  MoveL 2052 to (224.55, 431.71, -17.53) mm, rotated rx -180 ry 0 rz -11.91 deg; joints [23.109, -21.337, 64.711, -81.9, 97.908, 133.105]
  MoveL 2053 to (224.32, 431.8, -17.52) mm, rotated rx -180 ry 0 rz -11.91 deg; joints [23.101, -21.338, 64.711, -81.906, 97.902, 133.105]
  MoveL 2054 to (224.09, 431.88, -17.52) mm, rotated rx -180 ry 0 rz -11.91 deg; joints [23.094, -21.339, 64.715, -81.911, 97.897, 133.106]
  MoveL 2055 to (224.01, 431.9, -17.53) mm, rotated rx -180 ry 0 rz -11.91 deg; joints [23.091, -21.34, 64.716, -81.912, 97.895, 133.106]
  MoveL 2056 to (223.77, 431.95, -17.53) mm, rotated rx -180 ry 0 rz -11.91 deg; joints [23.084, -21.343, 64.723, -81.917, 97.889, 133.109]
  MoveL 2057 to (223.53, 431.98, -17.53) mm, rotated rx -180 ry 0 rz -11.91 deg; joints [23.076, -21.347, 64.733, -81.921, 97.883, 133.114]
  MoveL 2058 to (223.29, 431.99, -17.53) mm, rotated rx -180 ry 0 rz -11.91 deg; joints [23.069, -21.353, 64.745, -81.925, 97.877, 133.119]
  MoveL 2059 to (223.05, 431.99, -17.53) mm, rotated rx 180 ry 0 rz -11.91 deg; joints [23.062, -21.359, 64.759, -81.929, 97.871, 133.126]
  MoveL 2060 to (-164.9, 431.99, -17.53) mm, rotated rx 180 ry 0 rz -11.91 deg; joints [11.107, -28.262, 79.844, -90.307, 89.248, 140.713]
  MoveL 2061 to (-194.97, 431.99, -17.52) mm, rotated rx -180 ry 0 rz -11.91 deg; joints [10.122, -28.555, 80.501, -91.087, 88.643, 141.084]
  MoveL 2062 to (-195.47, 431.99, -17.53) mm, rotated rx -180 ry 0 rz -11.91 deg; joints [10.106, -28.56, 80.512, -91.1, 88.633, 141.09]
  Set speed (38.1 mm/s)
  MoveL 2063 to (-196.09, 432.77, -17.53) mm, rotated rx -180 ry 0 rz -11.91 deg; joints [10.081, -28.525, 80.435, -91.119, 88.617, 141.049]
  MoveL 2064 to (-195.65, 434.72, -17.53) mm, rotated rx 180 ry 0 rz -11.91 deg; joints [10.084, -28.417, 80.2, -91.113, 88.616, 140.922]
  MoveL 2065 to (-195.51, 435.34, -16.89) mm, rotated rx 180 ry 0 rz -11.91 deg; joints [10.084, -28.412, 80.132, -91.111, 88.615, 140.859]
  Set speed (100.0 mm/s)
  MoveL 2066 to (-195.51, 435.34, 34.53) mm, rotated rx -180 ry 0 rz -11.91 deg; joints [10.073, -30.771, 80.586, -91.073, 88.572, 138.953]
  MoveL 2067 to (-195.51, 435.34, 34.53) mm, rotated rx -180 ry 0 rz -11.91 deg; joints [10.073, -30.771, 80.586, -91.073, 88.572, 138.953]

--- program Machining (robot KUKA KR 30 HA) ---
  Smooth(1)
  Print: /'1001'
  Print: /''
  Print: /'Parallel1'
  Call SetTool(1)
  Call SetRPM(5000.0)
  Set speed (1000.0 mm/s)
  Set Ref.: Frame 4
  Set Tool: rc90 spindle mm
  Show rc90 spindle mm
  MoveJ 1 to (194.72, 277.93, 99.72) mm, rotated rx -149.92 ry 0.28 rz 179.52 deg; joints [9.071, -45.044, 108.371, -170.24, 63.004, 205.935]
  MoveL 2 to (194.72, 277.93, 99.72) mm, rotated rx -149.92 ry 0.28 rz 179.52 deg; joints [9.071, -45.044, 108.371, -170.24, 63.004, 205.935]
  MoveL 3 to (194.72, 227.8, 13.19) mm, rotated rx -149.92 ry 0.28 rz 179.52 deg; joints [11.04, -39.933, 106.924, -168.39, 66.758, 205.788]
  MoveL 4 to (194.72, 227.8, 13.19) mm, rotated rx -149.92 ry 0.28 rz 179.52 deg; joints [11.04, -39.933, 106.924, -168.39, 66.758, 205.788]
  Set speed (1000.0 mm/s)
  MoveL 5 to (194.72, 218.79, -2.36) mm, rotated rx -149.92 ry 0.28 rz 179.52 deg; joints [11.391, -38.991, 106.584, -168.061, 67.374, 205.777]
  Set speed (16.7 mm/s)
  MoveL 6 to (194.72, 209.92, -17.68) mm, rotated rx -149.92 ry 0.28 rz 179.52 deg; joints [11.737, -38.057, 106.224, -167.738, 67.963, 205.769]
  MoveL 7 to (193.72, 209.42, -18.55) mm, rotated rx -149.92 ry 0.28 rz 179.52 deg; joints [11.765, -38.04, 106.292, -167.716, 68.048, 205.778]
  MoveL 8 to (193.59, 214.43, -9.89) mm, rotated rx -149.92 ry 0.28 rz 179.52 deg; joints [11.57, -38.574, 106.51, -167.897, 67.725, 205.783]
  MoveL 9 to (193.59, 214.44, -9.88) mm, rotated rx -149.92 ry 0.28 rz 179.52 deg; joints [11.57, -38.574, 106.51, -167.898, 67.724, 205.783]
  Set speed (1000.0 mm/s)
  MoveL 10 to (193.59, 222.79, 4.53) mm, rotated rx -149.92 ry 0.28 rz 179.52 deg; joints [11.244, -39.451, 106.838, -168.202, 67.161, 205.791]
  MoveL 11 to (194.72, 224.52, 3.53) mm, rotated rx -149.92 ry 0.28 rz 179.52 deg; joints [11.169, -39.365, 106.757, -168.284, 67.16, 205.822]
  MoveL 12 to (194.72, 217.03, -9.4) mm, rotated rx -149.92 ry 0.28 rz 179.52 deg; joints [11.461, -38.579, 106.464, -168.011, 67.665, 205.814]
  Set speed (16.7 mm/s)
  MoveL 13 to (194.72, 211.65, -18.68) mm, rotated rx -149.92 ry 0.28 rz 179.52 deg; joints [11.671, -38.012, 106.243, -167.815, 68.02, 205.81]
  MoveC 14 to (194.43, 211.3, -19.3) mm, rotated rx -149.92 ry 0.28 rz 179.52 deg; joints [11.687, -37.985, 106.254, -167.8, 68.058, 205.812] to (193.72, 211.15, -19.55) mm, rotated rx -149.92 ry 0.28 rz 179.52 deg; joints [11.698, -37.995, 106.31, -167.792, 68.105, 205.818]
  MoveL 15 to (193.72, 211.15, -19.55) mm, rotated rx -149.92 ry 0.28 rz 179.52 deg; joints [11.698, -37.995, 106.31, -167.792, 68.105, 205.818]
  MoveL 16 to (193.49, 216.16, -10.9) mm, rotated rx -149.92 ry 0.28 rz 179.52 deg; joints [11.505, -38.533, 106.538, -167.974, 67.787, 205.824]
  MoveL 17 to (191.2, 216.16, -10.9) mm, rotated rx -149.92 ry 0.28 rz 179.52 deg; joints [11.523, -38.615, 106.74, -167.965, 67.905, 205.844]
  MoveC 18 to (190.5, 216.31, -10.64) mm, rotated rx -149.92 ry 0.28 rz 179.52 deg; joints [11.523, -38.656, 106.808, -167.967, 67.932, 205.85] to (190.2, 216.66, -10.03) mm, rotated rx -149.92 ry 0.28 rz 179.52 deg; joints [11.511, -38.704, 106.848, -167.979, 67.923, 205.853]
  MoveL 19 to (190.2, 216.66, -10.03) mm, rotated rx -149.92 ry 0.28 rz 179.52 deg; joints [11.511, -38.704, 106.848, -167.979, 67.923, 205.853]
  Set speed (1000.0 mm/s)
  MoveL 20 to (190.2, 224.52, 3.53) mm, rotated rx -149.92 ry 0.28 rz 179.52 deg; joints [11.204, -39.531, 107.156, -168.266, 67.392, 205.86]
  MoveL 21 to (-191.54, 222.79, 4.53) mm, rotated rx -149.92 ry 0.28 rz 179.52 deg; joints [15.261, -50.505, 137.346, -165.09, 86.292, 209.487]
  MoveL 22 to (-191.54, 219.49, -1.15) mm, rotated rx -149.92 ry 0.28 rz 179.52 deg; joints [15.432, -50.022, 137.196, -164.925, 86.617, 209.565]
  Set speed (16.7 mm/s)
  MoveL 23 to (-191.54, 214.63, -9.56) mm, rotated rx -149.92 ry 0.28 rz 179.52 deg; joints [15.684, -49.309, 136.968, -164.679, 87.087, 209.681]
  MoveL 24 to (-191.94, 214.43, -9.89) mm, rotated rx -149.92 ry 0.28 rz 179.52 deg; joints [15.699, -49.288, 136.987, -164.664, 87.126, 209.691]
  MoveL 25 to (-192.68, 214.43, -9.89) mm, rotated rx -149.92 ry 0.28 rz 179.52 deg; joints [15.71, -49.302, 137.04, -164.654, 87.164, 209.702]
  MoveL 26 to (-192.7, 209.42, -18.55) mm, rotated rx -149.92 ry 0.28 rz 179.52 deg; joints [15.969, -48.568, 136.797, -164.401, 87.639, 209.824]
  MoveL 27 to (-193.07, 211.15, -19.55) mm, rotated rx -149.92 ry 0.28 rz 179.52 deg; joints [15.887, -48.5, 136.842, -164.484, 87.747, 209.856]
  MoveL 28 to (-193.07, 216.16, -10.9) mm, rotated rx -149.92 ry 0.28 rz 179.52 deg; joints [15.628, -49.234, 137.086, -164.738, 87.273, 209.735]
  MoveL 29 to (-189.43, 216.16, -10.9) mm, rotated rx -149.92 ry 0.28 rz 179.52 deg; joints [15.576, -49.167, 136.825, -164.787, 87.086, 209.686]
  MoveL 30 to (-188.93, 216.41, -10.46) mm, rotated rx -149.92 ry 0.28 rz 179.52 deg; joints [15.556, -49.194, 136.801, -164.807, 87.037, 209.673]
  MoveC 31 to (-189.34, 217.09, -9.63) mm, rotated rx -149.92 ry 0.28 rz 179.52 deg; joints [15.527, -49.273, 136.858, -164.835, 87.014, 209.668] to (-190.32, 217.64, -9.44) mm, rotated rx -149.92 ry 0.28 rz 179.52 deg; joints [15.513, -49.309, 136.942, -164.851, 87.061, 209.682]
  MoveL 32 to (-190.32, 217.64, -9.44) mm, rotated rx -149.92 ry 0.28 rz 179.52 deg; joints [15.513, -49.309, 136.942, -164.851, 87.061, 209.682]
  MoveL 33 to (-192.56, 218.42, -9.89) mm, rotated rx -149.92 ry 0.28 rz 179.52 deg; joints [15.505, -49.318, 137.111, -164.86, 87.215, 209.724]
  MoveC 34 to (-193.55, 218.53, -10.47) mm, rotated rx -149.92 ry 0.28 rz 179.52 deg; joints [15.513, -49.289, 137.175, -164.853, 87.305, 209.748] to (-193.96, 218.14, -11.47) mm, rotated rx -149.92 ry 0.28 rz 179.52 deg; joints [15.54, -49.213, 137.18, -164.828, 87.384, 209.768]
  MoveL 35 to (-193.96, 218.14, -11.47) mm, rotated rx -149.92 ry 0.28 rz 179.52 deg; joints [15.54, -49.213, 137.18, -164.828, 87.384, 209.768]
  MoveL 36 to (-193.96, 213.13, -20.12) mm, rotated rx -149.92 ry 0.28 rz 179.52 deg; joints [15.799, -48.478, 136.935, -164.573, 87.859, 209.89]
  MoveL 37 to (-193.46, 212.88, -20.55) mm, rotated rx -149.92 ry 0.28 rz 179.52 deg; joints [15.805, -48.432, 136.887, -164.567, 87.856, 209.889]
  MoveL 38 to (-193.43, 217.89, -11.9) mm, rotated rx -149.92 ry 0.28 rz 179.52 deg; joints [15.545, -49.166, 137.131, -164.822, 87.381, 209.767]
  MoveL 39 to (193.49, 217.89, -11.9) mm, rotated rx -149.92 ry 0.28 rz 179.52 deg; joints [11.438, -38.488, 106.556, -168.051, 67.843, 205.865]
  MoveL 40 to (193.72, 212.88, -20.55) mm, rotated rx -149.92 ry 0.28 rz 179.52 deg; joints [11.632, -37.95, 106.328, -167.869, 68.161, 205.858]
  MoveL 41 to (193.72, 214.61, -21.55) mm, rotated rx -149.92 ry 0.28 rz 179.52 deg; joints [11.566, -37.905, 106.346, -167.945, 68.218, 205.898]
  MoveL 42 to (193.49, 219.62, -12.9) mm, rotated rx -149.92 ry 0.28 rz 179.52 deg; joints [11.372, -38.442, 106.574, -168.128, 67.9, 205.905]
  MoveL 43 to (-193.72, 219.62, -12.9) mm, rotated rx -149.92 ry 0.28 rz 179.52 deg; joints [15.461, -49.097, 137.169, -164.907, 87.485, 209.798]
  MoveL 44 to (-193.74, 214.61, -21.55) mm, rotated rx -149.92 ry 0.28 rz 179.52 deg; joints [15.721, -48.362, 136.925, -164.652, 87.96, 209.92]
  MoveL 45 to (-193.31, 216.34, -22.56) mm, rotated rx -149.92 ry 0.28 rz 179.52 deg; joints [15.627, -48.28, 136.912, -164.747, 88.026, 209.94]
  MoveL 46 to (-193.31, 221.35, -13.9) mm, rotated rx -149.92 ry 0.28 rz 179.52 deg; joints [15.367, -49.014, 137.158, -165.002, 87.552, 209.82]
  MoveL 47 to (193.28, 221.35, -13.9) mm, rotated rx -149.92 ry 0.28 rz 179.52 deg; joints [11.307, -38.405, 106.61, -168.204, 67.967, 205.947]
  MoveL 48 to (193.31, 216.34, -22.56) mm, rotated rx -149.92 ry 0.28 rz 179.52 deg; joints [11.502, -37.874, 106.399, -168.02, 68.295, 205.942]
  MoveL 49 to (191.75, 218.07, -23.56) mm, rotated rx -149.92 ry 0.28 rz 179.52 deg; joints [11.448, -37.884, 106.555, -168.09, 68.433, 205.995]
  MoveL 50 to (191.68, 223.08, -14.91) mm, rotated rx -149.92 ry 0.28 rz 179.52 deg; joints [11.253, -38.416, 106.768, -168.274, 68.107, 206]
  MoveL 51 to (-191.75, 223.08, -14.91) mm, rotated rx -149.92 ry 0.28 rz 179.52 deg; joints [15.257, -48.911, 137.063, -165.112, 87.56, 209.825]
  MoveL 52 to (-191.75, 218.07, -23.56) mm, rotated rx -149.92 ry 0.28 rz 179.52 deg; joints [15.517, -48.177, 136.817, -164.857, 88.033, 209.945]
  MoveC 53 to (-192.46, 218.22, -23.31) mm, rotated rx -149.92 ry 0.28 rz 179.52 deg; joints [15.519, -48.211, 136.875, -164.855, 88.056, 209.951] to (-192.75, 218.57, -22.69) mm, rotated rx -149.92 ry 0.28 rz 179.52 deg; joints [15.505, -48.268, 136.914, -164.869, 88.038, 209.947]
  MoveL 54 to (-192.75, 218.57, -22.69) mm, rotated rx -149.92 ry 0.28 rz 179.52 deg; joints [15.505, -48.268, 136.914, -164.869, 88.038, 209.947]
  Set speed (1000.0 mm/s)
  MoveL 55 to (-192.75, 236.46, 8.18) mm, rotated rx -149.92 ry 0.28 rz 179.52 deg; joints [14.575, -50.894, 137.748, -165.778, 86.296, 209.527]
  Print: /'Parallel2'
  Call SetTool(1)
  Call SetRPM(5000.0)
  Set speed (1000.0 mm/s)
  MoveL 56 to (-122.87, -170.47, 35.88) mm, rotated rx -149.92 ry 0.28 rz 179.52 deg; joints [31.344, -46.991, 120.44, -147.856, 75.214, 201.582]
  MoveL 57 to (-122.87, -192.28, -1.78) mm, rotated rx -149.92 ry 0.28 rz 179.52 deg; joints [32.175, -44.225, 119.07, -147.197, 76.514, 202.158]
  Set speed (16.7 mm/s)
  MoveL 58 to (-122.87, -206.58, -26.46) mm, rotated rx -149.92 ry 0.28 rz 179.52 deg; joints [32.712, -42.414, 118.095, -146.757, 77.289, 202.508]
  MoveC 59 to (-122.57, -206.94, -27.07) mm, rotated rx -149.92 ry 0.28 rz 179.52 deg; joints [32.718, -42.362, 118.05, -146.752, 77.296, 202.51] to (-121.87, -207.08, -27.32) mm, rotated rx -149.92 ry 0.28 rz 179.52 deg; joints [32.707, -42.325, 117.99, -146.76, 77.275, 202.5]
  MoveL 60 to (-121.87, -207.08, -27.32) mm, rotated rx -149.92 ry 0.28 rz 179.52 deg; joints [32.707, -42.325, 117.99, -146.76, 77.275, 202.5]
  MoveL 61 to (-121.78, -193.28, -3.5) mm, rotated rx -149.92 ry 0.28 rz 179.52 deg; joints [32.187, -44.069, 118.928, -147.186, 76.527, 202.162]
  MoveL 62 to (189.07, -193.28, -3.5) mm, rotated rx -149.92 ry 0.28 rz 179.52 deg; joints [26.181, -33.899, 94.323, -150.758, 62.981, 196.347]
  MoveL 63 to (189.08, -207.08, -27.32) mm, rotated rx -149.92 ry 0.28 rz 179.52 deg; joints [26.635, -32.401, 93.386, -150.403, 63.579, 196.439]
  MoveL 64 to (192.38, -208.45, -26.53) mm, rotated rx -149.92 ry 0.28 rz 179.52 deg; joints [26.626, -32.286, 93.034, -150.355, 63.37, 196.312]
  MoveL 65 to (193.72, -211.41, -24.82) mm, rotated rx -149.92 ry 0.28 rz 179.52 deg; joints [26.698, -32.266, 92.801, -150.224, 63.203, 196.16]
  MoveL 66 to (193.72, -197.6, -1) mm, rotated rx -149.92 ry 0.28 rz 179.52 deg; joints [26.246, -33.761, 93.74, -150.576, 62.609, 196.07]
  MoveL 67 to (-126.28, -197.6, -1) mm, rotated rx -149.92 ry 0.28 rz 179.52 deg; joints [32.45, -44.28, 119.084, -146.912, 76.518, 202.072]
  MoveL 68 to (-126.51, -211.41, -24.82) mm, rotated rx -149.92 ry 0.28 rz 179.52 deg; joints [32.973, -42.537, 118.157, -146.485, 77.273, 202.418]
  MoveL 69 to (-126.14, -213.57, -23.57) mm, rotated rx -149.92 ry 0.28 rz 179.52 deg; joints [33.042, -42.574, 118.051, -146.397, 77.164, 202.322]
  MoveL 70 to (-125.68, -215.73, -22.32) mm, rotated rx -149.92 ry 0.28 rz 179.52 deg; joints [33.109, -42.608, 117.94, -146.311, 77.053, 202.226]
  MoveL 71 to (-125.64, -207.44, -8.02) mm, rotated rx -149.92 ry 0.28 rz 179.52 deg; joints [32.799, -43.655, 118.509, -146.563, 76.611, 202.022]
  MoveL 72 to (-121.57, -207.44, -8.02) mm, rotated rx -149.92 ry 0.28 rz 179.52 deg; joints [32.703, -43.547, 118.225, -146.637, 76.45, 201.944]
  MoveL 73 to (-121.42, -201.93, 1.51) mm, rotated rx -149.92 ry 0.28 rz 179.52 deg; joints [32.494, -44.24, 118.584, -146.806, 76.139, 201.803]
  MoveL 74 to (188.78, -201.93, 1.51) mm, rotated rx -149.92 ry 0.28 rz 179.52 deg; joints [26.463, -34.003, 94.024, -150.349, 62.698, 195.987]
  MoveL 75 to (188.9, -207.44, -8.02) mm, rotated rx -149.92 ry 0.28 rz 179.52 deg; joints [26.642, -33.402, 93.646, -150.211, 62.937, 196.024]
  MoveL 76 to (193.72, -207.44, -8.02) mm, rotated rx -149.92 ry 0.28 rz 179.52 deg; joints [26.565, -33.21, 93.208, -150.232, 62.704, 195.925]
  MoveL 77 to (193.72, -215.73, -22.32) mm, rotated rx -149.92 ry 0.28 rz 179.52 deg; joints [26.835, -32.312, 92.638, -150.022, 63.055, 195.977]
  MoveL 78 to (193.72, -217.89, -21.07) mm, rotated rx -149.92 ry 0.28 rz 179.52 deg; joints [26.903, -32.334, 92.555, -149.921, 62.981, 195.885]
  MoveL 79 to (193.7, -220.05, -19.82) mm, rotated rx -149.92 ry 0.28 rz 179.52 deg; joints [26.972, -32.357, 92.474, -149.819, 62.908, 195.793]
  MoveL 80 to (193.7, -211.76, -5.52) mm, rotated rx -149.92 ry 0.28 rz 179.52 deg; joints [26.702, -33.255, 93.044, -150.028, 62.557, 195.74]
  MoveL 81 to (-124.73, -211.76, -5.52) mm, rotated rx -149.92 ry 0.28 rz 179.52 deg; joints [32.934, -43.72, 118.284, -146.388, 76.388, 201.827]
  MoveL 82 to (-124.77, -220.05, -19.82) mm, rotated rx -149.92 ry 0.28 rz 179.52 deg; joints [33.242, -42.674, 117.716, -146.138, 76.83, 202.031]
  MoveC 83 to (-125.47, -219.9, -19.56) mm, rotated rx -149.92 ry 0.28 rz 179.52 deg; joints [33.253, -42.711, 117.776, -146.129, 76.851, 202.041] to (-125.77, -219.55, -18.95) mm, rotated rx -149.92 ry 0.28 rz 179.52 deg; joints [33.247, -42.764, 117.821, -146.134, 76.844, 202.038]
  MoveL 84 to (-125.77, -219.55, -18.95) mm, rotated rx -149.92 ry 0.28 rz 179.52 deg; joints [33.247, -42.764, 117.821, -146.134, 76.844, 202.038]
  Set speed (1000.0 mm/s)
  MoveL 85 to (-125.77, -183.44, 43.39) mm, rotated rx -149.92 ry 0.28 rz 179.52 deg; joints [31.891, -47.334, 120.153, -147.206, 74.768, 201.093]
  Print: /'Contour6'
  Call SetTool(1)
  Call SetRPM(5000.0)
  Set speed (1000.0 mm/s)
  MoveL 86 to (-194.89, 224.1, 15) mm, rotated rx -180 ry 0 rz 179.9 deg; joints [21.967, -53.45, 134.896, -157.76, 81.141, 176.985]
  MoveL 87 to (-194.89, 224.1, 1.16) mm, rotated rx -180 ry 0 rz 179.9 deg; joints [21.974, -52.375, 134.756, -157.806, 82.007, 177.341]
  Set speed (5.6 mm/s)
  MoveL 88 to (-194.89, 224.1, -5) mm, rotated rx -180 ry 0 rz 179.9 deg; joints [21.977, -51.896, 134.688, -157.824, 82.388, 177.498]
  MoveC 89 to (-194.65, 223.92, -5.71) mm, rotated rx 180 ry 0 rz 179.9 deg; joints [21.981, -51.833, 134.658, -157.822, 82.418, 177.51] to (-194.08, 223.5, -6) mm, rotated rx -180 ry 0 rz 179.9 deg; joints [21.99, -51.793, 134.603, -157.812, 82.404, 177.503]
  Set speed (16.7 mm/s)
  MoveL 90 to (-190.41, 220.78, -6) mm, rotated rx 180 ry 0 rz 179.9 deg; joints [22.048, -51.682, 134.266, -157.742, 82.198, 177.41]
  MoveL 91 to (-190.31, 219.26, -6) mm, rotated rx 180 ry 0 rz 179.9 deg; joints [22.118, -51.666, 134.215, -157.67, 82.17, 177.388]
  MoveL 92 to (-190.6, 218.98, -6) mm, rotated rx -180 ry 0 rz 179.9 deg; joints [22.136, -51.67, 134.227, -157.651, 82.178, 177.389]
  MoveL 93 to (-190.82, 218.73, -6) mm, rotated rx 180 ry 0 rz 179.9 deg; joints [22.153, -51.673, 134.236, -157.635, 82.184, 177.389]
  MoveL 94 to (-191.02, 218.47, -6) mm, rotated rx 180 ry 0 rz 179.9 deg; joints [22.169, -51.676, 134.243, -157.619, 82.188, 177.389]
  MoveL 95 to (-191.23, 218.16, -6) mm, rotated rx -180 ry 0 rz 179.9 deg; joints [22.187, -51.678, 134.248, -157.601, 82.193, 177.388]
  MoveL 96 to (-191.4, 217.86, -6) mm, rotated rx 180 ry 0 rz 179.9 deg; joints [22.205, -51.679, 134.252, -157.583, 82.195, 177.387]
  MoveL 97 to (-191.55, 217.55, -6) mm, rotated rx 180 ry 0 rz 179.9 deg; joints [22.222, -51.68, 134.253, -157.565, 82.197, 177.385]
  MoveL 98 to (-191.68, 217.24, -6) mm, rotated rx -180 ry 0 rz 179.9 deg; joints [22.239, -51.68, 134.253, -157.549, 82.198, 177.383]
  MoveL 99 to (-191.78, 216.94, -6) mm, rotated rx -180 ry 0 rz 179.9 deg; joints [22.255, -51.68, 134.251, -157.532, 82.197, 177.38]
  MoveL 100 to (-191.86, 216.63, -6) mm, rotated rx 180 ry 0 rz 179.9 deg; joints [22.271, -51.679, 134.248, -157.516, 82.196, 177.377]
  MoveL 101 to (-191.91, 216.32, -6) mm, rotated rx 180 ry 0 rz 179.9 deg; joints [22.287, -51.678, 134.243, -157.5, 82.193, 177.374]
  MoveL 102 to (-191.95, 216.02, -6) mm, rotated rx 180 ry 0 rz 179.9 deg; joints [22.302, -51.676, 134.237, -157.484, 82.19, 177.371]
  MoveL 103 to (-191.97, 215.71, -6) mm, rotated rx -180 ry 0 rz 179.9 deg; joints [22.317, -51.674, 134.23, -157.469, 82.186, 177.367]
  MoveL 104 to (-191.98, 215.4, -6) mm, rotated rx 180 ry 0 rz 179.9 deg; joints [22.331, -51.671, 134.221, -157.454, 82.181, 177.363]
  MoveL 105 to (-191.98, 213.56, -6) mm, rotated rx -180 ry 0 rz 179.9 deg; joints [22.418, -51.654, 134.168, -157.365, 82.152, 177.338]
  MoveL 106 to (-191.97, 212.33, -6) mm, rotated rx -180 ry 0 rz 179.9 deg; joints [22.475, -51.643, 134.131, -157.306, 82.131, 177.321]
  MoveL 107 to (-191.94, 212.03, -6) mm, rotated rx 180 ry 0 rz 179.9 deg; joints [22.489, -51.639, 134.12, -157.292, 82.125, 177.317]
  MoveL 108 to (-191.89, 211.72, -6) mm, rotated rx 180 ry 0 rz 179.9 deg; joints [22.503, -51.635, 134.108, -157.278, 82.118, 177.312]
  MoveL 109 to (-126.45, -201.29, -6) mm, rotated rx 180 ry 0 rz 179.9 deg; joints [37.304, -43.646, 112.662, -140.567, 72.542, 167.063]
  MoveL 110 to (-126.38, -201.66, -6) mm, rotated rx 180 ry 0 rz 179.9 deg; joints [37.314, -43.636, 112.637, -140.554, 72.533, 167.05]
  MoveL 111 to (-126.27, -202.03, -6) mm, rotated rx 180 ry 0 rz 179.9 deg; joints [37.324, -43.625, 112.61, -140.541, 72.523, 167.037]
  MoveL 112 to (-126.2, -202.24, -6) mm, rotated rx -180 ry 0 rz 179.9 deg; joints [37.329, -43.618, 112.594, -140.534, 72.517, 167.029]
  MoveL 113 to (-126.11, -202.46, -6) mm, rotated rx 180 ry 0 rz 179.9 deg; joints [37.334, -43.611, 112.577, -140.527, 72.51, 167.021]
  MoveL 114 to (-126.02, -202.67, -6) mm, rotated rx 180 ry 0 rz 179.9 deg; joints [37.338, -43.604, 112.559, -140.52, 72.503, 167.013]
  MoveL 115 to (-125.91, -202.89, -6) mm, rotated rx 180 ry 0 rz 179.9 deg; joints [37.343, -43.596, 112.54, -140.513, 72.495, 167.004]
  MoveL 116 to (-125.78, -203.1, -6) mm, rotated rx 180 ry 0 rz 179.9 deg; joints [37.346, -43.588, 112.52, -140.507, 72.487, 166.995]
  MoveL 117 to (-125.64, -203.31, -6) mm, rotated rx -180 ry 0 rz 179.9 deg; joints [37.35, -43.579, 112.5, -140.501, 72.479, 166.986]
  MoveL 118 to (-125.49, -203.53, -6) mm, rotated rx -180 ry 0 rz 179.9 deg; joints [37.353, -43.57, 112.478, -140.495, 72.47, 166.977]
  MoveL 119 to (-125.32, -203.74, -6) mm, rotated rx -180 ry 0 rz 179.9 deg; joints [37.356, -43.56, 112.454, -140.49, 72.46, 166.967]
  MoveL 120 to (-125.14, -203.94, -6) mm, rotated rx 180 ry 0 rz 179.9 deg; joints [37.358, -43.551, 112.432, -140.485, 72.45, 166.958]
  MoveL 121 to (-124.94, -204.13, -6) mm, rotated rx -180 ry 0 rz 179.9 deg; joints [37.359, -43.541, 112.408, -140.481, 72.44, 166.948]
  MoveL 122 to (-124.76, -204.3, -6) mm, rotated rx 180 ry 0 rz 179.9 deg; joints [37.36, -43.532, 112.386, -140.478, 72.43, 166.939]
  MoveL 123 to (-124.57, -204.45, -6) mm, rotated rx -180 ry 0 rz 179.9 deg; joints [37.36, -43.523, 112.365, -140.475, 72.421, 166.931]
  MoveL 124 to (-124.2, -204.72, -6) mm, rotated rx 180 ry 0 rz 179.9 deg; joints [37.359, -43.506, 112.326, -140.471, 72.403, 166.916]
  MoveL 125 to (-123.82, -204.93, -6) mm, rotated rx 180 ry 0 rz 179.9 deg; joints [37.357, -43.491, 112.288, -140.469, 72.386, 166.902]
  MoveL 126 to (-123.52, -205.08, -6) mm, rotated rx 180 ry 0 rz 179.9 deg; joints [37.354, -43.479, 112.259, -140.468, 72.372, 166.892]
  MoveL 127 to (-123.21, -205.2, -6) mm, rotated rx 180 ry 0 rz 179.9 deg; joints [37.351, -43.467, 112.232, -140.469, 72.359, 166.882]
  MoveL 128 to (-122.9, -205.3, -6) mm, rotated rx 180 ry 0 rz 179.9 deg; joints [37.346, -43.456, 112.205, -140.47, 72.346, 166.873]
  MoveL 129 to (-122.6, -205.38, -6) mm, rotated rx 180 ry 0 rz 179.9 deg; joints [37.341, -43.445, 112.18, -140.473, 72.333, 166.865]
  MoveL 130 to (-122.29, -205.44, -6) mm, rotated rx -180 ry 0 rz 179.9 deg; joints [37.335, -43.435, 112.156, -140.476, 72.321, 166.857]
  MoveL 131 to (-121.98, -205.47, -6) mm, rotated rx 180 ry 0 rz 179.9 deg; joints [37.329, -43.425, 112.133, -140.479, 72.31, 166.85]
  MoveL 132 to (-121.37, -205.5, -6) mm, rotated rx 180 ry 0 rz 179.9 deg; joints [37.315, -43.407, 112.089, -140.489, 72.287, 166.838]
  MoveL 133 to (182.67, -205.5, -6) mm, rotated rx 180 ry 0 rz 179.9 deg; joints [30.898, -32.659, 87.872, -143.562, 59.81, 160.402]
  MoveL 134 to (188.8, -205.5, -6) mm, rotated rx 180 ry 0 rz 179.9 deg; joints [30.789, -32.398, 87.302, -143.573, 59.525, 160.248]
  MoveL 135 to (189.1, -205.48, -6) mm, rotated rx 180 ry 0 rz 179.9 deg; joints [30.783, -32.385, 87.274, -143.574, 59.511, 160.241]
  MoveL 136 to (189.41, -205.45, -6) mm, rotated rx 180 ry 0 rz 179.9 deg; joints [30.777, -32.373, 87.248, -143.576, 59.497, 160.234]
  MoveL 137 to (189.72, -205.4, -6) mm, rotated rx -180 ry 0 rz 179.9 deg; joints [30.77, -32.361, 87.222, -143.579, 59.484, 160.228]
  MoveL 138 to (190.02, -205.32, -6) mm, rotated rx -180 ry 0 rz 179.9 deg; joints [30.762, -32.349, 87.197, -143.583, 59.47, 160.223]
  MoveL 139 to (190.26, -205.25, -6) mm, rotated rx -180 ry 0 rz 179.9 deg; joints [30.756, -32.341, 87.179, -143.586, 59.46, 160.22]
  MoveL 140 to (190.64, -205.11, -6) mm, rotated rx 180 ry 0 rz 179.9 deg; joints [30.745, -32.328, 87.152, -143.593, 59.445, 160.215]
  MoveL 141 to (190.94, -204.97, -6) mm, rotated rx 180 ry 0 rz 179.9 deg; joints [30.736, -32.319, 87.131, -143.599, 59.432, 160.213]
  MoveL 142 to (191.25, -204.81, -6) mm, rotated rx -180 ry 0 rz 179.9 deg; joints [30.725, -32.31, 87.111, -143.607, 59.42, 160.211]
  MoveL 143 to (191.56, -204.61, -6) mm, rotated rx -180 ry 0 rz 179.9 deg; joints [30.714, -32.301, 87.094, -143.616, 59.409, 160.211]
  MoveL 144 to (191.86, -204.39, -6) mm, rotated rx 180 ry 0 rz 179.9 deg; joints [30.702, -32.294, 87.078, -143.626, 59.398, 160.211]
  MoveL 145 to (192.17, -204.12, -6) mm, rotated rx -180 ry 0 rz 179.9 deg; joints [30.689, -32.287, 87.064, -143.638, 59.388, 160.214]
  MoveL 146 to (192.33, -203.96, -6) mm, rotated rx 180 ry 0 rz 179.9 deg; joints [30.681, -32.285, 87.058, -143.645, 59.382, 160.216]
  MoveL 147 to (192.48, -203.8, -6) mm, rotated rx 180 ry 0 rz 179.9 deg; joints [30.674, -32.282, 87.053, -143.652, 59.378, 160.218]
  MoveL 148 to (192.52, -203.74, -6) mm, rotated rx 180 ry 0 rz 179.9 deg; joints [30.671, -32.282, 87.051, -143.655, 59.376, 160.219]
  MoveL 149 to (192.77, -203.43, -6) mm, rotated rx 180 ry 0 rz 179.9 deg; joints [30.658, -32.279, 87.046, -143.668, 59.369, 160.224]
  MoveL 150 to (192.97, -203.13, -6) mm, rotated rx -180 ry 0 rz 179.9 deg; joints [30.645, -32.278, 87.044, -143.682, 59.364, 160.23]
  MoveL 151 to (193.15, -202.82, -6) mm, rotated rx 180 ry 0 rz 179.9 deg; joints [30.633, -32.278, 87.044, -143.695, 59.361, 160.237]
  MoveL 152 to (193.29, -202.51, -6) mm, rotated rx 180 ry 0 rz 179.9 deg; joints [30.621, -32.279, 87.047, -143.709, 59.358, 160.245]
  MoveL 153 to (193.42, -202.21, -6) mm, rotated rx -180 ry 0 rz 179.9 deg; joints [30.61, -32.281, 87.053, -143.722, 59.357, 160.253]
  MoveL 154 to (193.52, -201.9, -6) mm, rotated rx 180 ry 0 rz 179.9 deg; joints [30.599, -32.285, 87.06, -143.736, 59.356, 160.262]
  MoveL 155 to (193.6, -201.59, -6) mm, rotated rx 180 ry 0 rz 179.9 deg; joints [30.589, -32.289, 87.07, -143.749, 59.357, 160.271]
  MoveL 156 to (193.66, -201.29, -6) mm, rotated rx -180 ry 0 rz 179.9 deg; joints [30.578, -32.294, 87.081, -143.762, 59.359, 160.281]
  MoveL 157 to (193.7, -200.98, -6) mm, rotated rx 180 ry 0 rz 179.9 deg; joints [30.569, -32.3, 87.095, -143.776, 59.362, 160.291]
  MoveL 158 to (193.72, -200.67, -6) mm, rotated rx -180 ry 0 rz 179.9 deg; joints [30.559, -32.307, 87.11, -143.789, 59.365, 160.302]
  MoveL 159 to (193.72, -200.06, -6) mm, rotated rx 180 ry 0 rz 179.9 deg; joints [30.541, -32.322, 87.144, -143.815, 59.374, 160.325]
  MoveL 160 to (193.72, 215.4, -6) mm, rotated rx 180 ry 0 rz 179.9 deg; joints [16.669, -39.631, 103.922, -161.48, 64.521, 172.291]
  MoveL 161 to (193.72, 215.71, -6) mm, rotated rx -180 ry 0 rz 179.9 deg; joints [16.658, -39.635, 103.93, -161.493, 64.524, 172.298]
  MoveL 162 to (193.7, 216.02, -6) mm, rotated rx 180 ry 0 rz 179.9 deg; joints [16.647, -39.639, 103.94, -161.506, 64.528, 172.305]
  MoveL 163 to (193.66, 216.32, -6) mm, rotated rx 180 ry 0 rz 179.9 deg; joints [16.636, -39.644, 103.952, -161.519, 64.533, 172.313]
  MoveL 164 to (193.6, 216.63, -6) mm, rotated rx 180 ry 0 rz 179.9 deg; joints [16.625, -39.649, 103.965, -161.531, 64.539, 172.32]
  MoveL 165 to (193.52, 216.94, -6) mm, rotated rx 180 ry 0 rz 179.9 deg; joints [16.615, -39.656, 103.981, -161.544, 64.546, 172.328]
  MoveL 166 to (193.42, 217.24, -6) mm, rotated rx -180 ry 0 rz 179.9 deg; joints [16.605, -39.663, 103.998, -161.557, 64.554, 172.336]
  MoveL 167 to (193.3, 217.55, -6) mm, rotated rx 180 ry 0 rz 179.9 deg; joints [16.595, -39.671, 104.017, -161.569, 64.563, 172.344]
  MoveL 168 to (193.15, 217.86, -6) mm, rotated rx 180 ry 0 rz 179.9 deg; joints [16.585, -39.68, 104.038, -161.582, 64.573, 172.353]
  MoveL 169 to (192.97, 218.16, -6) mm, rotated rx 180 ry 0 rz 179.9 deg; joints [16.576, -39.691, 104.062, -161.594, 64.585, 172.362]
  MoveL 170 to (192.77, 218.47, -6) mm, rotated rx -180 ry 0 rz 179.9 deg; joints [16.567, -39.702, 104.088, -161.606, 64.598, 172.371]
  MoveL 171 to (192.63, 218.65, -6) mm, rotated rx 180 ry 0 rz 179.9 deg; joints [16.562, -39.709, 104.105, -161.614, 64.606, 172.377]
  MoveL 172 to (192.48, 218.84, -6) mm, rotated rx 180 ry 0 rz 179.9 deg; joints [16.556, -39.717, 104.124, -161.621, 64.615, 172.383]
  MoveL 173 to (192.33, 219, -6) mm, rotated rx 180 ry 0 rz 179.9 deg; joints [16.552, -39.725, 104.141, -161.627, 64.624, 172.388]
  MoveL 174 to (192.17, 219.16, -6) mm, rotated rx 180 ry 0 rz 179.9 deg; joints [16.548, -39.733, 104.159, -161.633, 64.634, 172.394]
  MoveL 175 to (191.86, 219.42, -6) mm, rotated rx 180 ry 0 rz 179.9 deg; joints [16.542, -39.748, 104.194, -161.643, 64.651, 172.404]
  MoveL 176 to (191.56, 219.65, -6) mm, rotated rx 180 ry 0 rz 179.9 deg; joints [16.536, -39.762, 104.227, -161.651, 64.668, 172.413]
  MoveL 177 to (191.25, 219.85, -6) mm, rotated rx -180 ry 0 rz 179.9 deg; joints [16.533, -39.776, 104.259, -161.658, 64.685, 172.421]
  MoveL 178 to (190.94, 220.01, -6) mm, rotated rx -180 ry 0 rz 179.9 deg; joints [16.53, -39.789, 104.291, -161.664, 64.702, 172.428]
  MoveL 179 to (190.64, 220.15, -6) mm, rotated rx -180 ry 0 rz 179.9 deg; joints [16.528, -39.803, 104.322, -161.668, 64.718, 172.435]
  MoveL 180 to (190.33, 220.27, -6) mm, rotated rx 180 ry 0 rz 179.9 deg; joints [16.527, -39.816, 104.352, -161.672, 64.734, 172.441]
  MoveL 181 to (190.02, 220.36, -6) mm, rotated rx 180 ry 0 rz 179.9 deg; joints [16.527, -39.829, 104.381, -161.675, 64.75, 172.447]
  MoveL 182 to (189.72, 220.43, -6) mm, rotated rx 180 ry 0 rz 179.9 deg; joints [16.528, -39.841, 104.41, -161.676, 64.766, 172.453]
  MoveL 183 to (189.41, 220.49, -6) mm, rotated rx -180 ry 0 rz 179.9 deg; joints [16.529, -39.854, 104.439, -161.677, 64.781, 172.458]
  MoveL 184 to (189.1, 220.52, -6) mm, rotated rx 180 ry 0 rz 179.9 deg; joints [16.531, -39.866, 104.467, -161.677, 64.797, 172.462]
  MoveL 185 to (188.8, 220.53, -6) mm, rotated rx 180 ry 0 rz 179.9 deg; joints [16.534, -39.878, 104.494, -161.676, 64.812, 172.466]
  MoveL 186 to (187.57, 220.53, -6) mm, rotated rx -180 ry 0 rz 179.9 deg; joints [16.548, -39.925, 104.603, -161.67, 64.872, 172.481]
  MoveL 187 to (-186.96, 220.53, -6) mm, rotated rx -180 ry 0 rz 179.9 deg; joints [21.994, -51.597, 134.014, -157.788, 82.042, 177.353]
  MoveL 188 to (-187.26, 220.53, -6) mm, rotated rx 180 ry 0 rz 179.9 deg; joints [22, -51.604, 134.036, -157.782, 82.055, 177.358]
  MoveL 189 to (-187.57, 220.5, -6) mm, rotated rx 180 ry 0 rz 179.9 deg; joints [22.007, -51.611, 134.057, -157.776, 82.068, 177.362]
  MoveL 190 to (-187.88, 220.45, -6) mm, rotated rx 180 ry 0 rz 179.9 deg; joints [22.015, -51.618, 134.077, -157.768, 82.081, 177.366]
  MoveL 191 to (-188.18, 220.39, -6) mm, rotated rx -180 ry 0 rz 179.9 deg; joints [22.024, -51.625, 134.097, -157.76, 82.094, 177.37]
  MoveL 192 to (-188.49, 220.3, -6) mm, rotated rx -180 ry 0 rz 179.9 deg; joints [22.034, -51.631, 134.116, -157.751, 82.106, 177.374]
  MoveL 193 to (-188.8, 220.19, -6) mm, rotated rx -180 ry 0 rz 179.9 deg; joints [22.045, -51.638, 134.135, -157.74, 82.118, 177.377]
  MoveL 194 to (-189.1, 220.06, -6) mm, rotated rx 180 ry 0 rz 179.9 deg; joints [22.057, -51.644, 134.153, -157.729, 82.129, 177.38]
  MoveL 195 to (-189.41, 219.9, -6) mm, rotated rx -180 ry 0 rz 179.9 deg; joints [22.07, -51.65, 134.17, -157.716, 82.14, 177.383]
  MoveL 196 to (-189.72, 219.72, -6) mm, rotated rx 180 ry 0 rz 179.9 deg; joints [22.085, -51.656, 134.186, -157.702, 82.151, 177.385]
  MoveL 197 to (-190.02, 219.5, -6) mm, rotated rx 180 ry 0 rz 179.9 deg; joints [22.101, -51.661, 134.201, -157.686, 82.161, 177.387]
  MoveL 198 to (-190.31, 219.26, -6) mm, rotated rx 180 ry 0 rz 179.9 deg; joints [22.118, -51.666, 134.215, -157.67, 82.17, 177.388]
  MoveC 199 to (-191.1, 218.99, -6) mm, rotated rx -180 ry 0 rz 179.9 deg; joints [22.146, -51.682, 134.263, -157.643, 82.2, 177.397] to (-191.83, 219.41, -6) mm, rotated rx 180 ry 0 rz 179.9 deg; joints [22.14, -51.703, 134.326, -157.651, 82.239, 177.414]
  MoveL 200 to (-194.43, 223.17, -6) mm, rotated rx 180 ry 0 rz 179.9 deg; joints [22.013, -51.799, 134.617, -157.789, 82.414, 177.504]
  MoveC 201 to (-194.83, 223.75, -5.71) mm, rotated rx 180 ry 0 rz 179.9 deg; joints [21.993, -51.836, 134.666, -157.81, 82.423, 177.51] to (-195, 223.99, -5) mm, rotated rx -180 ry 0 rz 179.9 deg; joints [21.984, -51.897, 134.692, -157.817, 82.391, 177.498]
  Set speed (1000.0 mm/s)
  MoveL 202 to (-195, 223.99, 6) mm, rotated rx 180 ry 0 rz 179.9 deg; joints [21.979, -52.753, 134.812, -157.783, 81.709, 177.218]
  MoveL 203 to (176.9, -186.06, 6) mm, rotated rx 180 ry 0 rz 179.9 deg; joints [30.415, -33.959, 89.574, -144.226, 59.973, 160.932]
  MoveL 204 to (176.9, -186.06, 1.5) mm, rotated rx -180 ry 0 rz 179.9 deg; joints [30.416, -33.741, 89.535, -144.284, 60.119, 161.051]
  Set speed (5.6 mm/s)
  MoveL 205 to (176.9, -186.06, -5) mm, rotated rx -180 ry 0 rz 179.9 deg; joints [30.419, -33.425, 89.475, -144.367, 60.328, 161.222]
  MoveC 206 to (177.13, -186.24, -5.71) mm, rotated rx 180 ry 0 rz 179.9 deg; joints [30.421, -33.377, 89.437, -144.368, 60.337, 161.229] to (177.68, -186.68, -6) mm, rotated rx -180 ry 0 rz 179.9 deg; joints [30.424, -33.329, 89.36, -144.355, 60.314, 161.207]
  Set speed (16.7 mm/s)
  MoveL 207 to (183.64, -191.36, -6) mm, rotated rx 180 ry 0 rz 179.9 deg; joints [30.459, -32.965, 88.559, -144.17, 59.971, 160.894]
  MoveL 208 to (183.72, -192.46, -6) mm, rotated rx -180 ry 0 rz 179.9 deg; joints [30.491, -32.935, 88.492, -144.123, 59.951, 160.852]
  MoveL 209 to (183.59, -192.6, -6) mm, rotated rx 180 ry 0 rz 179.9 deg; joints [30.497, -32.937, 88.496, -144.117, 59.955, 160.85]
  MoveL 210 to (-117.09, -192.6, -6) mm, rotated rx 180 ry 0 rz 179.9 deg; joints [36.788, -43.556, 112.468, -141.074, 72.344, 167.145]
  MoveL 211 to (-117.27, -192.46, -6) mm, rotated rx -180 ry 0 rz 179.9 deg; joints [36.787, -43.564, 112.487, -141.076, 72.353, 167.152]
  MoveL 212 to (-180.63, 207.46, -6) mm, rotated rx 180 ry 0 rz 179.9 deg; joints [22.483, -51.324, 133.188, -157.264, 81.556, 177.077]
  MoveL 213 to (-180.41, 207.64, -6) mm, rotated rx 180 ry 0 rz 179.9 deg; joints [22.47, -51.32, 133.178, -157.276, 81.549, 177.076]
  MoveL 214 to (183.59, 207.64, -6) mm, rotated rx 180 ry 0 rz 179.9 deg; joints [17.069, -39.933, 104.609, -161.1, 64.941, 172.248]
  MoveL 215 to (183.72, 207.46, -6) mm, rotated rx -180 ry 0 rz 179.9 deg; joints [17.074, -39.926, 104.593, -161.093, 64.933, 172.242]
  MoveL 216 to (183.72, -192.46, -6) mm, rotated rx -180 ry 0 rz 179.9 deg; joints [30.491, -32.935, 88.492, -144.123, 59.951, 160.852]
  Set speed (5.6 mm/s)
  MoveL 217 to (183.72, -192.46, -12) mm, rotated rx 180 ry 0 rz 179.9 deg; joints [30.493, -32.643, 88.432, -144.199, 60.14, 161.008]
  Set speed (16.7 mm/s)
  MoveL 218 to (183.59, -192.6, -12) mm, rotated rx -180 ry 0 rz 179.9 deg; joints [30.5, -32.645, 88.437, -144.193, 60.144, 161.006]
  MoveL 219 to (-117.09, -192.6, -12) mm, rotated rx 180 ry 0 rz 179.9 deg; joints [36.791, -43.204, 112.409, -141.129, 72.573, 167.337]
  MoveL 220 to (-117.27, -192.46, -12) mm, rotated rx 180 ry 0 rz 179.9 deg; joints [36.79, -43.212, 112.428, -141.131, 72.582, 167.345]
  MoveL 221 to (-180.22, 204.81, -12) mm, rotated rx 180 ry 0 rz 179.9 deg; joints [22.6, -50.832, 133.012, -157.163, 81.853, 177.185]
  MoveL 222 to (-180.43, 206.2, -12) mm, rotated rx -180 ry 0 rz 179.9 deg; joints [22.54, -50.85, 133.068, -157.225, 81.885, 177.207]
  MoveL 223 to (-180.22, 206.4, -12) mm, rotated rx 180 ry 0 rz 179.9 deg; joints [22.527, -50.847, 133.058, -157.239, 81.878, 177.207]
  MoveL 224 to (183.59, 206.4, -12) mm, rotated rx -180 ry 0 rz 179.9 deg; joints [17.117, -39.591, 104.517, -161.086, 65.184, 172.316]
  MoveL 225 to (183.72, 206.2, -12) mm, rotated rx 180 ry 0 rz 179.9 deg; joints [17.123, -39.584, 104.5, -161.078, 65.176, 172.309]
  MoveL 226 to (183.72, -192.46, -12) mm, rotated rx 180 ry 0 rz 179.9 deg; joints [30.493, -32.643, 88.432, -144.199, 60.14, 161.008]
  Set speed (5.6 mm/s)
  MoveL 227 to (183.72, -192.46, -18) mm, rotated rx -180 ry 0 rz 179.9 deg; joints [30.495, -32.35, 88.37, -144.274, 60.328, 161.162]
  Set speed (16.7 mm/s)
  MoveL 228 to (183.59, -192.6, -18) mm, rotated rx -180 ry 0 rz 179.9 deg; joints [30.502, -32.353, 88.375, -144.267, 60.332, 161.16]
  MoveL 229 to (-117.09, -192.6, -18) mm, rotated rx 180 ry 0 rz 179.9 deg; joints [36.794, -42.85, 112.347, -141.183, 72.801, 167.528]
  MoveL 230 to (-117.27, -192.46, -18) mm, rotated rx 180 ry 0 rz 179.9 deg; joints [36.793, -42.858, 112.366, -141.185, 72.81, 167.536]
  MoveL 231 to (-180.22, 204.81, -18) mm, rotated rx 180 ry 0 rz 179.9 deg; joints [22.603, -50.375, 132.939, -157.181, 82.207, 177.335]
  MoveL 232 to (-180.43, 206.2, -18) mm, rotated rx -180 ry 0 rz 179.9 deg; joints [22.543, -50.393, 132.995, -157.243, 82.24, 177.357]
  MoveL 233 to (-180.22, 206.4, -18) mm, rotated rx 180 ry 0 rz 179.9 deg; joints [22.53, -50.389, 132.985, -157.257, 82.233, 177.357]
  MoveL 234 to (183.59, 206.4, -18) mm, rotated rx 180 ry 0 rz 179.9 deg; joints [17.119, -39.262, 104.456, -161.123, 65.438, 172.41]
  MoveL 235 to (183.72, 206.2, -18) mm, rotated rx -180 ry 0 rz 179.9 deg; joints [17.125, -39.255, 104.439, -161.115, 65.429, 172.404]
  MoveL 236 to (183.72, -192.46, -18) mm, rotated rx -180 ry 0 rz 179.9 deg; joints [30.495, -32.35, 88.37, -144.274, 60.328, 161.162]
  Set speed (5.6 mm/s)
  MoveL 237 to (183.72, -192.46, -20.05) mm, rotated rx 180 ry 0 rz 179.9 deg; joints [30.496, -32.25, 88.348, -144.299, 60.392, 161.215]
  Set speed (16.7 mm/s)
  MoveL 238 to (183.59, -192.6, -20.05) mm, rotated rx -180 ry 0 rz 179.9 deg; joints [30.503, -32.252, 88.353, -144.292, 60.396, 161.213]
  MoveL 239 to (-117.09, -192.6, -20.05) mm, rotated rx 180 ry 0 rz 179.9 deg; joints [36.795, -42.729, 112.325, -141.201, 72.879, 167.593]
  MoveL 240 to (-117.27, -192.46, -20.05) mm, rotated rx -180 ry 0 rz 179.9 deg; joints [36.795, -42.737, 112.344, -141.203, 72.888, 167.6]
  MoveL 241 to (-180.22, 204.81, -20.05) mm, rotated rx 180 ry 0 rz 179.9 deg; joints [22.604, -50.219, 132.913, -157.187, 82.328, 177.386]
  MoveL 242 to (-180.43, 206.2, -20.05) mm, rotated rx 180 ry 0 rz 179.9 deg; joints [22.544, -50.236, 132.969, -157.249, 82.36, 177.408]
  MoveL 243 to (-180.22, 206.4, -20.05) mm, rotated rx -180 ry 0 rz 179.9 deg; joints [22.531, -50.233, 132.96, -157.263, 82.354, 177.408]
  MoveL 244 to (183.59, 206.4, -20.05) mm, rotated rx -180 ry 0 rz 179.9 deg; joints [17.119, -39.15, 104.434, -161.136, 65.524, 172.442]
  MoveL 245 to (183.72, 206.2, -20.05) mm, rotated rx -180 ry 0 rz 179.9 deg; joints [17.125, -39.142, 104.417, -161.128, 65.515, 172.436]
  MoveL 246 to (183.72, -192.46, -20.05) mm, rotated rx 180 ry 0 rz 179.9 deg; joints [30.496, -32.25, 88.348, -144.299, 60.392, 161.215]
  Set speed (1000.0 mm/s)
  MoveL 247 to (183.72, -192.46, 6) mm, rotated rx -180 ry 0 rz 179.9 deg; joints [30.486, -33.514, 88.601, -143.968, 59.569, 160.535]
  MoveL 248 to (-122.54, -205.85, 6) mm, rotated rx 180 ry 0 rz 179.9 deg; joints [37.349, -44.133, 112.26, -140.34, 71.867, 166.455]
  MoveL 249 to (-122.54, -205.85, 5.17) mm, rotated rx -180 ry 0 rz 179.9 deg; joints [37.349, -44.085, 112.253, -140.348, 71.899, 166.483]
  Set speed (5.6 mm/s)
  MoveL 250 to (-122.54, -205.85, -4.96) mm, rotated rx -180 ry 0 rz 179.9 deg; joints [37.354, -43.494, 112.161, -140.445, 72.284, 166.816]
  Set speed (16.7 mm/s)
  MoveL 251 to (-122.46, -205.97, -5.48) mm, rotated rx -180 ry 0 rz 179.9 deg; joints [37.357, -43.459, 112.145, -140.447, 72.299, 166.827]
  MoveL 252 to (-122.4, -206.34, -5.86) mm, rotated rx 180 ry 0 rz 179.9 deg; joints [37.367, -43.427, 112.117, -140.437, 72.305, 166.827]
  MoveL 253 to (-122.65, -206.78, -6) mm, rotated rx 180 ry 0 rz 179.9 deg; joints [37.388, -43.417, 112.11, -140.416, 72.312, 166.823]
  MoveL 254 to (-123.23, -207.24, -6) mm, rotated rx -180 ry 0 rz 179.9 deg; joints [37.418, -43.424, 112.126, -140.388, 72.326, 166.82]
  MoveL 255 to (-123.55, -207.56, -6) mm, rotated rx -180 ry 0 rz 179.9 deg; joints [37.436, -43.426, 112.131, -140.37, 72.332, 166.817]
  MoveL 256 to (-123.82, -207.88, -6) mm, rotated rx 180 ry 0 rz 179.9 deg; joints [37.453, -43.427, 112.133, -140.353, 72.337, 166.812]
  MoveL 257 to (-124.09, -208.26, -6) mm, rotated rx 180 ry 0 rz 179.9 deg; joints [37.472, -43.427, 112.131, -140.333, 72.34, 166.806]
  MoveL 258 to (-124.31, -208.65, -6) mm, rotated rx -180 ry 0 rz 179.9 deg; joints [37.49, -43.425, 112.126, -140.314, 72.342, 166.798]
  MoveL 259 to (-124.46, -208.96, -6) mm, rotated rx 180 ry 0 rz 179.9 deg; joints [37.504, -43.423, 112.119, -140.299, 72.342, 166.792]
  MoveL 260 to (-124.58, -209.27, -6) mm, rotated rx -180 ry 0 rz 179.9 deg; joints [37.517, -43.419, 112.111, -140.285, 72.341, 166.785]
  MoveL 261 to (-124.67, -209.57, -6) mm, rotated rx -180 ry 0 rz 179.9 deg; joints [37.529, -43.416, 112.102, -140.271, 72.339, 166.777]
  MoveL 262 to (-124.75, -209.88, -6) mm, rotated rx 180 ry 0 rz 179.9 deg; joints [37.541, -43.411, 112.091, -140.257, 72.337, 166.769]
  MoveL 263 to (-124.78, -210.03, -6) mm, rotated rx 180 ry 0 rz 179.9 deg; joints [37.547, -43.409, 112.085, -140.251, 72.336, 166.765]
  MoveL 264 to (-124.81, -210.19, -6) mm, rotated rx 180 ry 0 rz 179.9 deg; joints [37.552, -43.406, 112.078, -140.244, 72.334, 166.761]
  MoveL 265 to (-124.83, -210.34, -6) mm, rotated rx 180 ry 0 rz 179.9 deg; joints [37.558, -43.403, 112.071, -140.238, 72.332, 166.757]
  MoveL 266 to (-124.84, -210.49, -6) mm, rotated rx -180 ry 0 rz 179.9 deg; joints [37.563, -43.401, 112.064, -140.232, 72.33, 166.752]
  MoveL 267 to (-124.85, -210.65, -6) mm, rotated rx 180 ry 0 rz 179.9 deg; joints [37.568, -43.398, 112.057, -140.225, 72.328, 166.748]
  MoveL 268 to (-124.86, -210.8, -6) mm, rotated rx 180 ry 0 rz 179.9 deg; joints [37.573, -43.394, 112.049, -140.219, 72.326, 166.743]
  MoveL 269 to (-124.86, -210.95, -6) mm, rotated rx -180 ry 0 rz 179.9 deg; joints [37.578, -43.391, 112.041, -140.213, 72.323, 166.738]
  MoveL 270 to (-124.86, -211.11, -6) mm, rotated rx 180 ry 0 rz 179.9 deg; joints [37.583, -43.388, 112.033, -140.207, 72.321, 166.734]
  MoveL 271 to (-124.85, -211.26, -6) mm, rotated rx 180 ry 0 rz 179.9 deg; joints [37.588, -43.384, 112.024, -140.201, 72.318, 166.729]
  MoveL 272 to (-124.84, -211.41, -6) mm, rotated rx 180 ry 0 rz 179.9 deg; joints [37.593, -43.381, 112.015, -140.195, 72.315, 166.724]
  MoveL 273 to (-124.82, -211.57, -6) mm, rotated rx -180 ry 0 rz 179.9 deg; joints [37.597, -43.377, 112.006, -140.19, 72.312, 166.719]
  MoveL 274 to (-124.8, -211.72, -6) mm, rotated rx 180 ry 0 rz 179.9 deg; joints [37.602, -43.373, 111.996, -140.184, 72.308, 166.714]
  MoveL 275 to (-124.7, -212.33, -6) mm, rotated rx 180 ry 0 rz 179.9 deg; joints [37.619, -43.356, 111.957, -140.162, 72.295, 166.693]
  MoveL 276 to (-124.64, -212.64, -6) mm, rotated rx 180 ry 0 rz 179.9 deg; joints [37.627, -43.348, 111.936, -140.15, 72.287, 166.682]
  MoveL 277 to (-124.56, -212.95, -6) mm, rotated rx 180 ry 0 rz 179.9 deg; joints [37.635, -43.339, 111.914, -140.14, 72.279, 166.671]
  MoveL 278 to (-124.45, -213.25, -6) mm, rotated rx -180 ry 0 rz 179.9 deg; joints [37.643, -43.329, 111.891, -140.13, 72.27, 166.66]
  MoveL 279 to (-124.33, -213.56, -6) mm, rotated rx -180 ry 0 rz 179.9 deg; joints [37.649, -43.319, 111.866, -140.12, 72.261, 166.648]
  MoveL 280 to (-124.22, -213.78, -6) mm, rotated rx 180 ry 0 rz 179.9 deg; joints [37.654, -43.311, 111.847, -140.113, 72.253, 166.639]
  MoveL 281 to (-124.1, -214, -6) mm, rotated rx -180 ry 0 rz 179.9 deg; joints [37.658, -43.303, 111.827, -140.106, 72.245, 166.63]
  MoveL 282 to (-123.97, -214.22, -6) mm, rotated rx -180 ry 0 rz 179.9 deg; joints [37.662, -43.294, 111.806, -140.1, 72.237, 166.621]
  MoveL 283 to (-123.82, -214.43, -6) mm, rotated rx 180 ry 0 rz 179.9 deg; joints [37.665, -43.285, 111.784, -140.094, 72.228, 166.612]
  MoveL 284 to (-123.63, -214.68, -6) mm, rotated rx 180 ry 0 rz 179.9 deg; joints [37.668, -43.274, 111.758, -140.088, 72.217, 166.6]
  MoveL 285 to (-123.41, -214.93, -6) mm, rotated rx -180 ry 0 rz 179.9 deg; joints [37.671, -43.262, 111.729, -140.082, 72.205, 166.588]
  MoveL 286 to (-123.14, -215.19, -6) mm, rotated rx 180 ry 0 rz 179.9 deg; joints [37.673, -43.248, 111.697, -140.076, 72.191, 166.575]
  MoveL 287 to (-122.87, -215.42, -6) mm, rotated rx 180 ry 0 rz 179.9 deg; joints [37.673, -43.235, 111.666, -140.071, 72.177, 166.563]
  MoveL 288 to (-122.64, -215.6, -6) mm, rotated rx -180 ry 0 rz 179.9 deg; joints [37.673, -43.224, 111.64, -140.069, 72.165, 166.553]
  MoveL 289 to (-122.4, -215.76, -6) mm, rotated rx 180 ry 0 rz 179.9 deg; joints [37.672, -43.214, 111.615, -140.067, 72.154, 166.543]
  MoveL 290 to (-122.16, -215.89, -6) mm, rotated rx 180 ry 0 rz 179.9 deg; joints [37.671, -43.204, 111.591, -140.065, 72.143, 166.534]
  MoveL 291 to (-121.92, -216.02, -6) mm, rotated rx 180 ry 0 rz 179.9 deg; joints [37.669, -43.194, 111.569, -140.064, 72.133, 166.526]
  MoveL 292 to (-121.65, -216.14, -6) mm, rotated rx 180 ry 0 rz 179.9 deg; joints [37.666, -43.184, 111.543, -140.064, 72.121, 166.517]
  MoveL 293 to (-121.37, -216.24, -6) mm, rotated rx 180 ry 0 rz 179.9 deg; joints [37.662, -43.173, 111.518, -140.065, 72.109, 166.508]
  MoveL 294 to (-121.06, -216.33, -6) mm, rotated rx -180 ry 0 rz 179.9 deg; joints [37.657, -43.162, 111.492, -140.067, 72.096, 166.5]
  MoveL 295 to (-120.76, -216.41, -6) mm, rotated rx 180 ry 0 rz 179.9 deg; joints [37.652, -43.151, 111.467, -140.069, 72.084, 166.492]
  MoveL 296 to (-120.45, -216.46, -6) mm, rotated rx -180 ry 0 rz 179.9 deg; joints [37.646, -43.141, 111.443, -140.072, 72.072, 166.484]
  MoveL 297 to (-120.14, -216.49, -6) mm, rotated rx 180 ry 0 rz 179.9 deg; joints [37.639, -43.131, 111.42, -140.076, 72.06, 166.477]
  MoveL 298 to (-118.92, -216.5, -6) mm, rotated rx -180 ry 0 rz 179.9 deg; joints [37.609, -43.095, 111.334, -140.097, 72.015, 166.453]
  MoveL 299 to (182.67, -216.5, -6) mm, rotated rx 180 ry 0 rz 179.9 deg; joints [31.224, -32.383, 87.256, -143.089, 59.649, 159.993]
  MoveL 300 to (188.8, -216.5, -6) mm, rotated rx -180 ry 0 rz 179.9 deg; joints [31.115, -32.12, 86.684, -143.099, 59.364, 159.837]
  MoveL 301 to (189.1, -216.49, -6) mm, rotated rx 180 ry 0 rz 179.9 deg; joints [31.109, -32.108, 86.657, -143.1, 59.35, 159.829]
  MoveL 302 to (189.41, -216.46, -6) mm, rotated rx -180 ry 0 rz 179.9 deg; joints [31.102, -32.095, 86.63, -143.102, 59.336, 159.823]
  MoveL 303 to (189.72, -216.4, -6) mm, rotated rx 180 ry 0 rz 179.9 deg; joints [31.095, -32.083, 86.604, -143.104, 59.323, 159.817]
  MoveL 304 to (190.02, -216.33, -6) mm, rotated rx 180 ry 0 rz 179.9 deg; joints [31.088, -32.072, 86.579, -143.108, 59.309, 159.812]
  MoveL 305 to (190.45, -216.2, -6) mm, rotated rx 180 ry 0 rz 179.9 deg; joints [31.076, -32.057, 86.547, -143.114, 59.291, 159.806]
  MoveL 306 to (190.87, -216.02, -6) mm, rotated rx 180 ry 0 rz 179.9 deg; joints [31.063, -32.043, 86.517, -143.123, 59.274, 159.802]
  MoveL 307 to (191.27, -215.8, -6) mm, rotated rx 180 ry 0 rz 179.9 deg; joints [31.05, -32.032, 86.492, -143.132, 59.259, 159.799]
  MoveL 308 to (191.47, -215.68, -6) mm, rotated rx 180 ry 0 rz 179.9 deg; joints [31.043, -32.026, 86.48, -143.138, 59.251, 159.799]
  MoveL 309 to (191.67, -215.54, -6) mm, rotated rx 180 ry 0 rz 179.9 deg; joints [31.035, -32.021, 86.469, -143.144, 59.244, 159.799]
  MoveL 310 to (191.87, -215.38, -6) mm, rotated rx -180 ry 0 rz 179.9 deg; joints [31.027, -32.016, 86.459, -143.151, 59.237, 159.8]
  MoveL 311 to (192.07, -215.21, -6) mm, rotated rx 180 ry 0 rz 179.9 deg; joints [31.018, -32.012, 86.45, -143.159, 59.23, 159.801]
  MoveL 312 to (192.29, -215.01, -6) mm, rotated rx -180 ry 0 rz 179.9 deg; joints [31.008, -32.008, 86.442, -143.168, 59.223, 159.803]
  MoveL 313 to (192.48, -214.81, -6) mm, rotated rx 180 ry 0 rz 179.9 deg; joints [30.999, -32.005, 86.435, -143.177, 59.217, 159.806]
  MoveL 314 to (192.73, -214.49, -6) mm, rotated rx -180 ry 0 rz 179.9 deg; joints [30.985, -32.002, 86.429, -143.191, 59.21, 159.811]
  MoveL 315 to (192.94, -214.18, -6) mm, rotated rx 180 ry 0 rz 179.9 deg; joints [30.973, -32.001, 86.427, -143.204, 59.204, 159.817]
  MoveL 316 to (193.12, -213.87, -6) mm, rotated rx 180 ry 0 rz 179.9 deg; joints [30.96, -32.001, 86.427, -143.218, 59.2, 159.824]
  MoveL 317 to (193.28, -213.56, -6) mm, rotated rx -180 ry 0 rz 179.9 deg; joints [30.948, -32.002, 86.43, -143.232, 59.198, 159.832]
  MoveL 318 to (193.4, -213.25, -6) mm, rotated rx -180 ry 0 rz 179.9 deg; joints [30.937, -32.004, 86.436, -143.245, 59.196, 159.84]
  MoveL 319 to (193.51, -212.95, -6) mm, rotated rx -180 ry 0 rz 179.9 deg; joints [30.926, -32.008, 86.443, -143.259, 59.196, 159.849]
  MoveL 320 to (193.59, -212.64, -6) mm, rotated rx 180 ry 0 rz 179.9 deg; joints [30.916, -32.012, 86.453, -143.272, 59.196, 159.859]
  MoveL 321 to (193.65, -212.33, -6) mm, rotated rx 180 ry 0 rz 179.9 deg; joints [30.905, -32.017, 86.464, -143.285, 59.198, 159.869]
  MoveL 322 to (193.69, -212.03, -6) mm, rotated rx -180 ry 0 rz 179.9 deg; joints [30.896, -32.023, 86.478, -143.299, 59.201, 159.879]
  MoveL 323 to (193.72, -211.72, -6) mm, rotated rx 180 ry 0 rz 179.9 deg; joints [30.886, -32.03, 86.493, -143.312, 59.204, 159.89]
  MoveL 324 to (193.72, -211.11, -6) mm, rotated rx 180 ry 0 rz 179.9 deg; joints [30.868, -32.045, 86.527, -143.338, 59.213, 159.913]
  MoveL 325 to (193.72, -210.8, -6) mm, rotated rx 180 ry 0 rz 179.9 deg; joints [30.859, -32.053, 86.544, -143.352, 59.217, 159.925]
  MoveL 326 to (193.71, -210.65, -6) mm, rotated rx -180 ry 0 rz 179.9 deg; joints [30.855, -32.057, 86.554, -143.358, 59.22, 159.931]
  MoveL 327 to (193.7, -210.49, -6) mm, rotated rx -180 ry 0 rz 179.9 deg; joints [30.85, -32.061, 86.563, -143.365, 59.223, 159.937]
  MoveL 328 to (193.69, -210.34, -6) mm, rotated rx 180 ry 0 rz 179.9 deg; joints [30.846, -32.066, 86.573, -143.372, 59.226, 159.943]
  MoveL 329 to (193.67, -210.19, -6) mm, rotated rx -180 ry 0 rz 179.9 deg; joints [30.842, -32.071, 86.584, -143.378, 59.229, 159.949]
  MoveL 330 to (193.64, -210.03, -6) mm, rotated rx 180 ry 0 rz 179.9 deg; joints [30.838, -32.076, 86.595, -143.385, 59.232, 159.955]
  MoveL 331 to (193.61, -209.88, -6) mm, rotated rx -180 ry 0 rz 179.9 deg; joints [30.834, -32.081, 86.607, -143.391, 59.236, 159.962]
  MoveL 332 to (193.57, -209.73, -6) mm, rotated rx 180 ry 0 rz 179.9 deg; joints [30.83, -32.086, 86.618, -143.398, 59.24, 159.969]
  MoveL 333 to (193.53, -209.57, -6) mm, rotated rx -180 ry 0 rz 179.9 deg; joints [30.826, -32.092, 86.631, -143.405, 59.244, 159.975]
  MoveL 334 to (193.49, -209.42, -6) mm, rotated rx -180 ry 0 rz 179.9 deg; joints [30.822, -32.098, 86.644, -143.411, 59.248, 159.982]
  MoveL 335 to (193.44, -209.27, -6) mm, rotated rx 180 ry 0 rz 179.9 deg; joints [30.819, -32.104, 86.657, -143.418, 59.253, 159.989]
  MoveL 336 to (193.38, -209.11, -6) mm, rotated rx 180 ry 0 rz 179.9 deg; joints [30.815, -32.11, 86.671, -143.424, 59.258, 159.997]
  MoveL 337 to (193.32, -208.96, -6) mm, rotated rx 180 ry 0 rz 179.9 deg; joints [30.812, -32.117, 86.686, -143.431, 59.263, 160.004]
  MoveL 338 to (193.25, -208.8, -6) mm, rotated rx -180 ry 0 rz 179.9 deg; joints [30.808, -32.123, 86.701, -143.437, 59.269, 160.011]
  MoveL 339 to (193.17, -208.65, -6) mm, rotated rx 180 ry 0 rz 179.9 deg; joints [30.805, -32.131, 86.716, -143.444, 59.274, 160.019]
  MoveL 340 to (193.03, -208.4, -6) mm, rotated rx 180 ry 0 rz 179.9 deg; joints [30.8, -32.143, 86.744, -143.455, 59.285, 160.032]
  MoveL 341 to (192.87, -208.14, -6) mm, rotated rx -180 ry 0 rz 179.9 deg; joints [30.795, -32.156, 86.774, -143.466, 59.296, 160.046]
  MoveL 342 to (192.69, -207.88, -6) mm, rotated rx -180 ry 0 rz 179.9 deg; joints [30.791, -32.171, 86.805, -143.476, 59.308, 160.06]
  MoveL 343 to (192.48, -207.63, -6) mm, rotated rx 180 ry 0 rz 179.9 deg; joints [30.787, -32.186, 86.839, -143.487, 59.322, 160.075]
  MoveL 344 to (192.21, -207.35, -6) mm, rotated rx 180 ry 0 rz 179.9 deg; joints [30.784, -32.205, 86.88, -143.499, 59.339, 160.093]
  MoveL 345 to (191.94, -207.1, -6) mm, rotated rx 180 ry 0 rz 179.9 deg; joints [30.781, -32.223, 86.919, -143.509, 59.355, 160.108]
  MoveL 346 to (191.67, -206.89, -6) mm, rotated rx -180 ry 0 rz 179.9 deg; joints [30.78, -32.239, 86.956, -143.518, 59.37, 160.123]
  MoveL 347 to (191.4, -206.71, -6) mm, rotated rx 180 ry 0 rz 179.9 deg; joints [30.779, -32.255, 86.991, -143.525, 59.385, 160.137]
  MoveL 348 to (190.87, -206.41, -6) mm, rotated rx -180 ry 0 rz 179.9 deg; joints [30.78, -32.286, 87.057, -143.537, 59.415, 160.161]
  MoveL 349 to (190.33, -206.2, -6) mm, rotated rx 180 ry 0 rz 179.9 deg; joints [30.783, -32.314, 87.12, -143.546, 59.443, 160.183]
  MoveL 350 to (190.26, -206.17, -6) mm, rotated rx 180 ry 0 rz 179.9 deg; joints [30.783, -32.318, 87.128, -143.547, 59.447, 160.186]
  MoveL 351 to (190.02, -206.1, -6) mm, rotated rx 180 ry 0 rz 179.9 deg; joints [30.785, -32.33, 87.154, -143.549, 59.459, 160.194]
  MoveL 352 to (189.72, -206.03, -6) mm, rotated rx -180 ry 0 rz 179.9 deg; joints [30.789, -32.345, 87.187, -143.552, 59.474, 160.205]
  MoveL 353 to (189.41, -205.98, -6) mm, rotated rx -180 ry 0 rz 179.9 deg; joints [30.793, -32.359, 87.218, -143.554, 59.489, 160.215]
  MoveL 354 to (189.1, -205.94, -6) mm, rotated rx 180 ry 0 rz 179.9 deg; joints [30.797, -32.373, 87.249, -143.554, 59.504, 160.224]
  MoveL 355 to (188.8, -205.93, -6) mm, rotated rx -180 ry 0 rz 179.9 deg; joints [30.802, -32.387, 87.278, -143.555, 59.519, 160.232]
  MoveL 356 to (187.57, -205.93, -6) mm, rotated rx 180 ry 0 rz 179.9 deg; joints [30.824, -32.439, 87.392, -143.552, 59.576, 160.263]
  MoveL 357 to (-118.92, -205.93, -6) mm, rotated rx -180 ry 0 rz 179.9 deg; joints [37.268, -43.325, 111.896, -140.514, 72.19, 166.777]
  MoveL 358 to (-120.14, -205.94, -6) mm, rotated rx 180 ry 0 rz 179.9 deg; joints [37.298, -43.361, 111.981, -140.493, 72.235, 166.801]
  MoveL 359 to (-120.76, -206.01, -6) mm, rotated rx -180 ry 0 rz 179.9 deg; joints [37.316, -43.377, 112.019, -140.479, 72.256, 166.81]
  MoveL 360 to (-121.37, -206.16, -6) mm, rotated rx -180 ry 0 rz 179.9 deg; joints [37.336, -43.392, 112.054, -140.463, 72.276, 166.817]
  MoveL 361 to (-121.47, -206.2, -6) mm, rotated rx 180 ry 0 rz 179.9 deg; joints [37.34, -43.395, 112.059, -140.46, 72.279, 166.818]
  MoveL 362 to (-122.06, -206.44, -6) mm, rotated rx -180 ry 0 rz 179.9 deg; joints [37.362, -43.407, 112.087, -140.44, 72.296, 166.822]
  MoveL 363 to (-122.65, -206.78, -6) mm, rotated rx 180 ry 0 rz 179.9 deg; joints [37.388, -43.417, 112.11, -140.416, 72.312, 166.823]
  MoveC 364 to (-123.38, -206.98, -6) mm, rotated rx 180 ry 0 rz 179.9 deg; joints [37.413, -43.434, 112.15, -140.395, 72.336, 166.831] to (-124.05, -206.61, -6) mm, rotated rx 180 ry 0 rz 179.9 deg; joints [37.417, -43.461, 112.216, -140.399, 72.366, 166.855]
  MoveL 365 to (-124.96, -206.23, -6) mm, rotated rx 180 ry 0 rz 179.9 deg; joints [37.428, -43.496, 112.298, -140.398, 72.405, 166.884]
  MoveL 366 to (-128.18, -206.64, -6) mm, rotated rx -180 ry 0 rz 179.9 deg; joints [37.522, -43.582, 112.499, -140.325, 72.515, 166.934]
  Set speed (5.6 mm/s)
  MoveL 367 to (-128.18, -206.64, -11) mm, rotated rx -180 ry 0 rz 179.9 deg; joints [37.524, -43.288, 112.449, -140.371, 72.705, 167.097]
  MoveC 368 to (-127.89, -206.6, -11.71) mm, rotated rx 180 ry 0 rz 179.9 deg; joints [37.516, -43.239, 112.425, -140.385, 72.721, 167.116] to (-127.19, -206.49, -12) mm, rotated rx 180 ry 0 rz 179.9 deg; joints [37.495, -43.203, 112.38, -140.404, 72.709, 167.115]
  Set speed (16.7 mm/s)
  MoveC 369 to (-126.45, -206.66, -12) mm, rotated rx 180 ry 0 rz 179.9 deg; joints [37.482, -43.178, 112.319, -140.41, 72.679, 167.095] to (-126.05, -207.32, -12) mm, rotated rx 180 ry 0 rz 179.9 deg; joints [37.493, -43.153, 112.257, -140.392, 72.653, 167.067]
  MoveL 370 to (-125.06, -213.56, -12) mm, rotated rx 180 ry 0 rz 179.9 deg; joints [37.671, -42.989, 111.857, -140.163, 72.512, 166.858]
  MoveL 371 to (-124.66, -216.02, -12) mm, rotated rx -180 ry 0 rz 179.9 deg; joints [37.74, -42.925, 111.699, -140.073, 72.456, 166.775]
  MoveL 372 to (-124.61, -216.25, -12) mm, rotated rx 180 ry 0 rz 179.9 deg; joints [37.746, -42.918, 111.682, -140.065, 72.45, 166.766]
  MoveL 373 to (-124.54, -216.49, -12) mm, rotated rx 180 ry 0 rz 179.9 deg; joints [37.752, -42.911, 111.665, -140.057, 72.444, 166.758]
  MoveL 374 to (-124.46, -216.73, -12) mm, rotated rx -180 ry 0 rz 179.9 deg; joints [37.758, -42.903, 111.647, -140.049, 72.437, 166.749]
  MoveL 375 to (-124.36, -216.96, -12) mm, rotated rx -180 ry 0 rz 179.9 deg; joints [37.763, -42.895, 111.627, -140.041, 72.429, 166.739]
  MoveL 376 to (-124.25, -217.2, -12) mm, rotated rx 180 ry 0 rz 179.9 deg; joints [37.768, -42.887, 111.607, -140.034, 72.421, 166.73]
  MoveL 377 to (-124.13, -217.44, -12) mm, rotated rx 180 ry 0 rz 179.9 deg; joints [37.772, -42.878, 111.586, -140.027, 72.413, 166.72]
  MoveL 378 to (-123.98, -217.67, -12) mm, rotated rx -180 ry 0 rz 179.9 deg; joints [37.776, -42.869, 111.563, -140.02, 72.403, 166.71]
  MoveL 379 to (-123.82, -217.91, -12) mm, rotated rx -180 ry 0 rz 179.9 deg; joints [37.78, -42.859, 111.54, -140.014, 72.394, 166.7]
  MoveL 380 to (-123.6, -218.19, -12) mm, rotated rx 180 ry 0 rz 179.9 deg; joints [37.784, -42.847, 111.509, -140.006, 72.381, 166.687]
  MoveL 381 to (-123.35, -218.47, -12) mm, rotated rx 180 ry 0 rz 179.9 deg; joints [37.786, -42.833, 111.477, -140, 72.367, 166.673]
  MoveL 382 to (-123.1, -218.71, -12) mm, rotated rx 180 ry 0 rz 179.9 deg; joints [37.788, -42.821, 111.447, -139.995, 72.354, 166.661]
  MoveL 383 to (-122.85, -218.91, -12) mm, rotated rx 180 ry 0 rz 179.9 deg; joints [37.788, -42.809, 111.419, -139.991, 72.342, 166.65]
  MoveL 384 to (-122.61, -219.1, -12) mm, rotated rx -180 ry 0 rz 179.9 deg; joints [37.788, -42.798, 111.392, -139.988, 72.329, 166.639]
  MoveL 385 to (-122.36, -219.26, -12) mm, rotated rx -180 ry 0 rz 179.9 deg; joints [37.787, -42.787, 111.366, -139.986, 72.318, 166.63]
  MoveL 386 to (-122.11, -219.4, -12) mm, rotated rx -180 ry 0 rz 179.9 deg; joints [37.785, -42.777, 111.342, -139.985, 72.306, 166.62]
  MoveL 387 to (-121.86, -219.52, -12) mm, rotated rx 180 ry 0 rz 179.9 deg; joints [37.783, -42.767, 111.318, -139.984, 72.295, 166.612]
  MoveL 388 to (-121.62, -219.63, -12) mm, rotated rx 180 ry 0 rz 179.9 deg; joints [37.78, -42.757, 111.295, -139.984, 72.285, 166.604]
  MoveL 389 to (-121.37, -219.72, -12) mm, rotated rx -180 ry 0 rz 179.9 deg; joints [37.777, -42.748, 111.273, -139.985, 72.274, 166.596]
  MoveL 390 to (-121.06, -219.81, -12) mm, rotated rx 180 ry 0 rz 179.9 deg; joints [37.772, -42.737, 111.247, -139.987, 72.261, 166.587]
  MoveL 391 to (-120.76, -219.88, -12) mm, rotated rx -180 ry 0 rz 179.9 deg; joints [37.767, -42.726, 111.222, -139.989, 72.249, 166.579]
  MoveL 392 to (-120.45, -219.93, -12) mm, rotated rx 180 ry 0 rz 179.9 deg; joints [37.761, -42.716, 111.198, -139.993, 72.237, 166.571]
  MoveL 393 to (-120.14, -219.97, -12) mm, rotated rx 180 ry 0 rz 179.9 deg; joints [37.754, -42.707, 111.175, -139.997, 72.225, 166.564]
  MoveL 394 to (-118.92, -219.98, -12) mm, rotated rx 180 ry 0 rz 179.9 deg; joints [37.724, -42.67, 111.089, -140.017, 72.18, 166.54]
  MoveL 395 to (182.67, -219.98, -12) mm, rotated rx -180 ry 0 rz 179.9 deg; joints [31.329, -32.006, 87, -143.017, 59.783, 160.022]
  MoveL 396 to (188.8, -219.98, -12) mm, rotated rx -180 ry 0 rz 179.9 deg; joints [31.219, -31.744, 86.428, -143.027, 59.496, 159.864]
  MoveL 397 to (189.1, -219.96, -12) mm, rotated rx 180 ry 0 rz 179.9 deg; joints [31.213, -31.731, 86.4, -143.028, 59.482, 159.857]
  MoveL 398 to (189.41, -219.93, -12) mm, rotated rx 180 ry 0 rz 179.9 deg; joints [31.207, -31.719, 86.373, -143.03, 59.468, 159.85]
  MoveL 399 to (189.72, -219.88, -12) mm, rotated rx 180 ry 0 rz 179.9 deg; joints [31.2, -31.707, 86.347, -143.033, 59.455, 159.844]
  MoveL 400 to (190.02, -219.81, -12) mm, rotated rx 180 ry 0 rz 179.9 deg; joints [31.192, -31.695, 86.322, -143.036, 59.442, 159.839]
  MoveL 401 to (190.31, -219.72, -12) mm, rotated rx -180 ry 0 rz 179.9 deg; joints [31.185, -31.685, 86.301, -143.041, 59.429, 159.835]
  MoveL 402 to (190.59, -219.62, -12) mm, rotated rx 180 ry 0 rz 179.9 deg; joints [31.177, -31.676, 86.28, -143.045, 59.418, 159.831]
  MoveL 403 to (190.88, -219.49, -12) mm, rotated rx 180 ry 0 rz 179.9 deg; joints [31.168, -31.667, 86.26, -143.051, 59.406, 159.829]
  MoveL 404 to (191.16, -219.34, -12) mm, rotated rx 180 ry 0 rz 179.9 deg; joints [31.158, -31.658, 86.242, -143.058, 59.395, 159.827]
  MoveL 405 to (191.45, -219.17, -12) mm, rotated rx 180 ry 0 rz 179.9 deg; joints [31.148, -31.65, 86.225, -143.066, 59.384, 159.826]
  MoveL 406 to (191.73, -218.97, -12) mm, rotated rx 180 ry 0 rz 179.9 deg; joints [31.137, -31.643, 86.209, -143.075, 59.374, 159.826]
  MoveL 407 to (192.02, -218.74, -12) mm, rotated rx 180 ry 0 rz 179.9 deg; joints [31.125, -31.637, 86.196, -143.085, 59.364, 159.828]
  MoveL 408 to (192.3, -218.47, -12) mm, rotated rx -180 ry 0 rz 179.9 deg; joints [31.112, -31.631, 86.184, -143.097, 59.355, 159.83]
  MoveL 409 to (192.48, -218.28, -12) mm, rotated rx 180 ry 0 rz 179.9 deg; joints [31.104, -31.629, 86.179, -143.105, 59.349, 159.833]
  MoveL 410 to (192.71, -218, -12) mm, rotated rx 180 ry 0 rz 179.9 deg; joints [31.091, -31.626, 86.173, -143.118, 59.342, 159.838]
  MoveL 411 to (192.91, -217.71, -12) mm, rotated rx 180 ry 0 rz 179.9 deg; joints [31.079, -31.624, 86.17, -143.13, 59.337, 159.843]
  MoveL 412 to (193.08, -217.43, -12) mm, rotated rx 180 ry 0 rz 179.9 deg; joints [31.068, -31.624, 86.17, -143.143, 59.333, 159.849]
  MoveL 413 to (193.23, -217.15, -12) mm, rotated rx -180 ry 0 rz 179.9 deg; joints [31.057, -31.625, 86.172, -143.155, 59.331, 159.856]
  MoveL 414 to (193.35, -216.87, -12) mm, rotated rx 180 ry 0 rz 179.9 deg; joints [31.047, -31.627, 86.177, -143.168, 59.329, 159.864]
  MoveL 415 to (193.46, -216.58, -12) mm, rotated rx -180 ry 0 rz 179.9 deg; joints [31.036, -31.629, 86.183, -143.18, 59.328, 159.871]
  MoveL 416 to (193.54, -216.3, -12) mm, rotated rx -180 ry 0 rz 179.9 deg; joints [31.026, -31.633, 86.191, -143.192, 59.328, 159.88]
  MoveL 417 to (193.61, -216.02, -12) mm, rotated rx 180 ry 0 rz 179.9 deg; joints [31.017, -31.637, 86.2, -143.205, 59.329, 159.889]
  MoveL 418 to (193.67, -215.71, -12) mm, rotated rx 180 ry 0 rz 179.9 deg; joints [31.007, -31.643, 86.212, -143.218, 59.331, 159.899]
  MoveL 419 to (193.7, -215.4, -12) mm, rotated rx -180 ry 0 rz 179.9 deg; joints [30.997, -31.649, 86.227, -143.231, 59.334, 159.91]
  MoveL 420 to (193.72, -215.09, -12) mm, rotated rx 180 ry 0 rz 179.9 deg; joints [30.988, -31.656, 86.242, -143.245, 59.338, 159.921]
  MoveL 421 to (193.72, -214.79, -12) mm, rotated rx 180 ry 0 rz 179.9 deg; joints [30.979, -31.664, 86.26, -143.258, 59.342, 159.932]
  MoveL 422 to (193.72, 217.86, -12) mm, rotated rx 180 ry 0 rz 179.9 deg; joints [16.581, -39.332, 103.929, -161.622, 64.799, 172.438]
  MoveL 423 to (193.72, 218.16, -12) mm, rotated rx 180 ry 0 rz 179.9 deg; joints [16.569, -39.336, 103.937, -161.635, 64.802, 172.445]
  MoveL 424 to (193.71, 218.32, -12) mm, rotated rx -180 ry 0 rz 179.9 deg; joints [16.564, -39.337, 103.941, -161.642, 64.804, 172.449]
  MoveL 425 to (193.7, 218.47, -12) mm, rotated rx 180 ry 0 rz 179.9 deg; joints [16.558, -39.339, 103.946, -161.648, 64.806, 172.452]
  MoveL 426 to (193.69, 218.62, -12) mm, rotated rx 180 ry 0 rz 179.9 deg; joints [16.553, -39.342, 103.952, -161.655, 64.808, 172.456]
  MoveL 427 to (193.67, 218.78, -12) mm, rotated rx 180 ry 0 rz 179.9 deg; joints [16.547, -39.344, 103.958, -161.661, 64.811, 172.459]
  MoveL 428 to (193.65, 218.93, -12) mm, rotated rx -180 ry 0 rz 179.9 deg; joints [16.542, -39.347, 103.964, -161.668, 64.813, 172.463]
  MoveL 429 to (193.62, 219.08, -12) mm, rotated rx 180 ry 0 rz 179.9 deg; joints [16.537, -39.35, 103.97, -161.674, 64.816, 172.467]
  MoveL 430 to (193.58, 219.24, -12) mm, rotated rx 180 ry 0 rz 179.9 deg; joints [16.531, -39.353, 103.978, -161.681, 64.82, 172.47]
  MoveL 431 to (193.54, 219.39, -12) mm, rotated rx -180 ry 0 rz 179.9 deg; joints [16.526, -39.356, 103.985, -161.687, 64.823, 172.474]
  MoveL 432 to (193.5, 219.54, -12) mm, rotated rx 180 ry 0 rz 179.9 deg; joints [16.521, -39.359, 103.993, -161.693, 64.827, 172.478]
  MoveL 433 to (193.45, 219.7, -12) mm, rotated rx 180 ry 0 rz 179.9 deg; joints [16.516, -39.363, 104.002, -161.7, 64.831, 172.482]
  MoveL 434 to (193.39, 219.85, -12) mm, rotated rx -180 ry 0 rz 179.9 deg; joints [16.511, -39.367, 104.011, -161.706, 64.835, 172.486]
  MoveL 435 to (193.33, 220, -12) mm, rotated rx 180 ry 0 rz 179.9 deg; joints [16.506, -39.371, 104.02, -161.712, 64.839, 172.49]
  MoveL 436 to (193.26, 220.16, -12) mm, rotated rx 180 ry 0 rz 179.9 deg; joints [16.501, -39.375, 104.03, -161.718, 64.844, 172.495]
  MoveL 437 to (193.19, 220.31, -12) mm, rotated rx 180 ry 0 rz 179.9 deg; joints [16.496, -39.38, 104.041, -161.725, 64.849, 172.499]
  MoveL 438 to (193.02, 220.62, -12) mm, rotated rx -180 ry 0 rz 179.9 deg; joints [16.487, -39.389, 104.064, -161.737, 64.861, 172.508]
  MoveL 439 to (192.82, 220.92, -12) mm, rotated rx 180 ry 0 rz 179.9 deg; joints [16.477, -39.4, 104.089, -161.749, 64.873, 172.517]
  MoveL 440 to (192.66, 221.15, -12) mm, rotated rx 180 ry 0 rz 179.9 deg; joints [16.471, -39.409, 104.11, -161.758, 64.883, 172.524]
  MoveL 441 to (192.48, 221.37, -12) mm, rotated rx -180 ry 0 rz 179.9 deg; joints [16.465, -39.418, 104.132, -161.766, 64.895, 172.531]
  MoveL 442 to (192.17, 221.69, -12) mm, rotated rx 180 ry 0 rz 179.9 deg; joints [16.457, -39.434, 104.168, -161.779, 64.913, 172.542]
  MoveL 443 to (191.86, 221.96, -12) mm, rotated rx 180 ry 0 rz 179.9 deg; joints [16.45, -39.448, 104.202, -161.789, 64.931, 172.551]
  MoveL 444 to (191.56, 222.19, -12) mm, rotated rx 180 ry 0 rz 179.9 deg; joints [16.445, -39.463, 104.235, -161.797, 64.948, 172.56]
  MoveL 445 to (191.25, 222.38, -12) mm, rotated rx -180 ry 0 rz 179.9 deg; joints [16.441, -39.476, 104.267, -161.804, 64.965, 172.568]
  MoveL 446 to (190.64, 222.69, -12) mm, rotated rx 180 ry 0 rz 179.9 deg; joints [16.436, -39.503, 104.33, -161.814, 64.998, 172.583]
  MoveL 447 to (190.02, 222.89, -12) mm, rotated rx 180 ry 0 rz 179.9 deg; joints [16.435, -39.529, 104.389, -161.82, 65.03, 172.595]
  MoveL 448 to (189.41, 223.02, -12) mm, rotated rx 180 ry 0 rz 179.9 deg; joints [16.438, -39.554, 104.447, -161.822, 65.062, 172.605]
  MoveL 449 to (188.8, 223.07, -12) mm, rotated rx 180 ry 0 rz 179.9 deg; joints [16.443, -39.578, 104.502, -161.822, 65.092, 172.614]
  MoveL 450 to (187.57, 223.07, -12) mm, rotated rx 180 ry 0 rz 179.9 deg; joints [16.456, -39.624, 104.611, -161.816, 65.153, 172.629]
  MoveL 451 to (-187.57, 223.07, -12) mm, rotated rx 180 ry 0 rz 179.9 deg; joints [21.889, -51.17, 134.06, -157.917, 82.474, 177.545]
  MoveL 452 to (-188.8, 223.05, -12) mm, rotated rx -180 ry 0 rz 179.9 deg; joints [21.913, -51.199, 134.146, -157.896, 82.528, 177.564]
  MoveL 453 to (-189.41, 222.96, -12) mm, rotated rx 180 ry 0 rz 179.9 deg; joints [21.929, -51.212, 134.187, -157.881, 82.554, 177.573]
  MoveL 454 to (-190.02, 222.79, -12) mm, rotated rx -180 ry 0 rz 179.9 deg; joints [21.949, -51.225, 134.225, -157.863, 82.579, 177.58]
  MoveL 455 to (-190.64, 222.53, -12) mm, rotated rx -180 ry 0 rz 179.9 deg; joints [21.973, -51.237, 134.261, -157.84, 82.602, 177.586]
  MoveL 456 to (-191.25, 222.17, -12) mm, rotated rx -180 ry 0 rz 179.9 deg; joints [22.002, -51.248, 134.294, -157.811, 82.623, 177.591]
  MoveL 457 to (-191.56, 221.94, -12) mm, rotated rx -180 ry 0 rz 179.9 deg; joints [22.019, -51.254, 134.309, -157.795, 82.633, 177.593]
  MoveL 458 to (-191.86, 221.66, -12) mm, rotated rx -180 ry 0 rz 179.9 deg; joints [22.037, -51.258, 134.323, -157.777, 82.643, 177.595]
  MoveL 459 to (-192.2, 221.3, -12) mm, rotated rx -180 ry 0 rz 179.9 deg; joints [22.061, -51.263, 134.336, -157.753, 82.652, 177.595]
  MoveL 460 to (-192.47, 220.95, -12) mm, rotated rx 180 ry 0 rz 179.9 deg; joints [22.083, -51.266, 134.346, -157.731, 82.658, 177.595]
  MoveL 461 to (-192.49, 220.92, -12) mm, rotated rx -180 ry 0 rz 179.9 deg; joints [22.084, -51.267, 134.346, -157.73, 82.659, 177.595]
  MoveL 462 to (-192.69, 220.62, -12) mm, rotated rx 180 ry 0 rz 179.9 deg; joints [22.102, -51.268, 134.351, -157.712, 82.662, 177.594]
  MoveL 463 to (-192.86, 220.31, -12) mm, rotated rx 180 ry 0 rz 179.9 deg; joints [22.12, -51.27, 134.354, -157.694, 82.665, 177.593]
  MoveL 464 to (-193, 220, -12) mm, rotated rx 180 ry 0 rz 179.9 deg; joints [22.137, -51.27, 134.355, -157.677, 82.666, 177.591]
  MoveL 465 to (-193.11, 219.7, -12) mm, rotated rx 180 ry 0 rz 179.9 deg; joints [22.154, -51.27, 134.355, -157.66, 82.666, 177.589]
  MoveL 466 to (-193.21, 219.39, -12) mm, rotated rx -180 ry 0 rz 179.9 deg; joints [22.17, -51.27, 134.353, -157.643, 82.666, 177.587]
  MoveL 467 to (-193.28, 219.08, -12) mm, rotated rx -180 ry 0 rz 179.9 deg; joints [22.186, -51.269, 134.349, -157.627, 82.664, 177.584]
  MoveL 468 to (-193.31, 218.93, -12) mm, rotated rx -180 ry 0 rz 179.9 deg; joints [22.194, -51.268, 134.347, -157.619, 82.663, 177.582]
  MoveL 469 to (-193.34, 218.78, -12) mm, rotated rx 180 ry 0 rz 179.9 deg; joints [22.202, -51.268, 134.344, -157.612, 82.661, 177.581]
  MoveL 470 to (-193.36, 218.62, -12) mm, rotated rx 180 ry 0 rz 179.9 deg; joints [22.209, -51.267, 134.341, -157.604, 82.66, 177.579]
  MoveL 471 to (-193.37, 218.47, -12) mm, rotated rx -180 ry 0 rz 179.9 deg; joints [22.217, -51.266, 134.338, -157.596, 82.658, 177.577]
  MoveL 472 to (-193.38, 218.32, -12) mm, rotated rx 180 ry 0 rz 179.9 deg; joints [22.224, -51.265, 134.334, -157.588, 82.656, 177.575]
  MoveL 473 to (-193.39, 218.16, -12) mm, rotated rx -180 ry 0 rz 179.9 deg; joints [22.232, -51.263, 134.33, -157.581, 82.653, 177.573]
  MoveL 474 to (-193.39, 218.01, -12) mm, rotated rx 180 ry 0 rz 179.9 deg; joints [22.239, -51.262, 134.325, -157.574, 82.651, 177.571]
  MoveL 475 to (-193.38, 217.86, -12) mm, rotated rx -180 ry 0 rz 179.9 deg; joints [22.246, -51.261, 134.321, -157.566, 82.648, 177.569]
  MoveL 476 to (-193.37, 217.7, -12) mm, rotated rx 180 ry 0 rz 179.9 deg; joints [22.253, -51.259, 134.316, -157.559, 82.645, 177.567]
  MoveL 477 to (-193.36, 217.55, -12) mm, rotated rx -180 ry 0 rz 179.9 deg; joints [22.26, -51.257, 134.31, -157.552, 82.642, 177.565]
  MoveL 478 to (-193.34, 217.4, -12) mm, rotated rx -180 ry 0 rz 179.9 deg; joints [22.267, -51.256, 134.305, -157.545, 82.639, 177.563]
  MoveL 479 to (-193.32, 217.24, -12) mm, rotated rx 180 ry 0 rz 179.9 deg; joints [22.274, -51.254, 134.299, -157.538, 82.635, 177.56]
  MoveL 480 to (-192.47, 211.92, -12) mm, rotated rx -180 ry 0 rz 179.9 deg; joints [22.508, -51.187, 134.085, -157.295, 82.51, 177.477]
  MoveL 481 to (-126.12, -206.86, -12) mm, rotated rx 180 ry 0 rz 179.9 deg; joints [37.48, -43.164, 112.286, -140.408, 72.664, 167.083]
  MoveL 482 to (-126.05, -207.32, -12) mm, rotated rx 180 ry 0 rz 179.9 deg; joints [37.493, -43.153, 112.257, -140.392, 72.653, 167.067]
  MoveC 483 to (-126.68, -208.41, -12) mm, rotated rx 180 ry 0 rz 179.9 deg; joints [37.544, -43.147, 112.242, -140.338, 72.658, 167.047] to (-127.87, -208.02, -12) mm, rotated rx -180 ry 0 rz 179.9 deg; joints [37.562, -43.19, 112.345, -140.332, 72.708, 167.082]
  MoveL 484 to (-128.72, -206.73, -12) mm, rotated rx -180 ry 0 rz 179.9 deg; joints [37.541, -43.243, 112.472, -140.368, 72.76, 167.137]
  Set speed (5.6 mm/s)
  MoveL 485 to (-128.72, -206.73, -17) mm, rotated rx 180 ry 0 rz 179.9 deg; joints [37.544, -42.948, 112.42, -140.413, 72.948, 167.299]
  MoveC 486 to (-128.43, -206.68, -17.71) mm, rotated rx 180 ry 0 rz 179.9 deg; joints [37.535, -42.899, 112.395, -140.426, 72.965, 167.317] to (-127.73, -206.57, -18) mm, rotated rx -180 ry 0 rz 179.9 deg; joints [37.514, -42.863, 112.35, -140.446, 72.953, 167.316]
  Set speed (16.7 mm/s)
  MoveC 487 to (-126.98, -206.75, -18) mm, rotated rx -180 ry 0 rz 179.9 deg; joints [37.502, -42.838, 112.289, -140.452, 72.922, 167.296] to (-126.58, -207.4, -18) mm, rotated rx 180 ry 0 rz 179.9 deg; joints [37.513, -42.813, 112.227, -140.433, 72.897, 167.269]
  MoveL 488 to (-124.73, -219.08, -18) mm, rotated rx 180 ry 0 rz 179.9 deg; joints [37.844, -42.509, 111.478, -140.007, 72.629, 166.875]
  MoveL 489 to (-124.68, -219.39, -18) mm, rotated rx 180 ry 0 rz 179.9 deg; joints [37.852, -42.501, 111.458, -139.996, 72.622, 166.865]
  MoveL 490 to (-124.61, -219.7, -18) mm, rotated rx 180 ry 0 rz 179.9 deg; joints [37.86, -42.493, 111.437, -139.985, 72.614, 166.854]
  MoveL 491 to (-124.52, -220, -18) mm, rotated rx -180 ry 0 rz 179.9 deg; joints [37.868, -42.484, 111.414, -139.975, 72.606, 166.843]
  MoveL 492 to (-124.41, -220.31, -18) mm, rotated rx 180 ry 0 rz 179.9 deg; joints [37.875, -42.474, 111.39, -139.964, 72.596, 166.831]
  MoveL 493 to (-124.28, -220.62, -18) mm, rotated rx -180 ry 0 rz 179.9 deg; joints [37.882, -42.463, 111.364, -139.955, 72.586, 166.819]
  MoveL 494 to (-124.12, -220.92, -18) mm, rotated rx 180 ry 0 rz 179.9 deg; joints [37.887, -42.452, 111.336, -139.946, 72.575, 166.806]
  MoveL 495 to (-123.98, -221.16, -18) mm, rotated rx 180 ry 0 rz 179.9 deg; joints [37.891, -42.443, 111.314, -139.939, 72.566, 166.796]
  MoveL 496 to (-123.82, -221.39, -18) mm, rotated rx -180 ry 0 rz 179.9 deg; joints [37.895, -42.433, 111.291, -139.933, 72.556, 166.786]
  MoveL 497 to (-123.69, -221.56, -18) mm, rotated rx -180 ry 0 rz 179.9 deg; joints [37.897, -42.426, 111.273, -139.928, 72.549, 166.778]
  MoveL 498 to (-123.54, -221.74, -18) mm, rotated rx 180 ry 0 rz 179.9 deg; joints [37.899, -42.418, 111.253, -139.924, 72.54, 166.77]
  MoveL 499 to (-123.38, -221.91, -18) mm, rotated rx -180 ry 0 rz 179.9 deg; joints [37.901, -42.409, 111.233, -139.92, 72.531, 166.761]
  MoveL 500 to (-123.21, -222.09, -18) mm, rotated rx 180 ry 0 rz 179.9 deg; joints [37.902, -42.4, 111.211, -139.916, 72.522, 166.752]
  MoveL 501 to (-122.9, -222.35, -18) mm, rotated rx -180 ry 0 rz 179.9 deg; joints [37.903, -42.386, 111.176, -139.911, 72.506, 166.738]
  MoveL 502 to (-122.6, -222.58, -18) mm, rotated rx -180 ry 0 rz 179.9 deg; joints [37.902, -42.372, 111.142, -139.907, 72.491, 166.725]
  MoveL 503 to (-122.29, -222.77, -18) mm, rotated rx 180 ry 0 rz 179.9 deg; joints [37.901, -42.359, 111.111, -139.905, 72.477, 166.713]
  MoveL 504 to (-121.98, -222.94, -18) mm, rotated rx 180 ry 0 rz 179.9 deg; joints [37.899, -42.346, 111.081, -139.904, 72.463, 166.702]
  MoveL 505 to (-121.68, -223.08, -18) mm, rotated rx 180 ry 0 rz 179.9 deg; joints [37.895, -42.334, 111.052, -139.904, 72.449, 166.691]
  MoveL 506 to (-121.37, -223.19, -18) mm, rotated rx 180 ry 0 rz 179.9 deg; joints [37.891, -42.323, 111.025, -139.905, 72.436, 166.682]
  MoveL 507 to (-121, -223.3, -18) mm, rotated rx 180 ry 0 rz 179.9 deg; joints [37.886, -42.31, 110.993, -139.907, 72.421, 166.671]
  MoveL 508 to (-120.63, -223.38, -18) mm, rotated rx 180 ry 0 rz 179.9 deg; joints [37.879, -42.297, 110.964, -139.91, 72.406, 166.661]
  MoveL 509 to (-120.2, -223.44, -18) mm, rotated rx -180 ry 0 rz 179.9 deg; joints [37.87, -42.284, 110.931, -139.915, 72.389, 166.651]
  MoveL 510 to (-119.78, -223.45, -18) mm, rotated rx -180 ry 0 rz 179.9 deg; joints [37.86, -42.271, 110.9, -139.922, 72.373, 166.642]
  MoveL 511 to (188.58, -223.45, -18) mm, rotated rx 180 ry 0 rz 179.9 deg; joints [31.328, -31.375, 86.187, -142.955, 59.636, 159.896]
  MoveL 512 to (189.08, -223.44, -18) mm, rotated rx 180 ry 0 rz 179.9 deg; joints [31.318, -31.354, 86.141, -142.956, 59.613, 159.883]
  MoveL 513 to (189.33, -223.42, -18) mm, rotated rx -180 ry 0 rz 179.9 deg; joints [31.313, -31.344, 86.119, -142.957, 59.602, 159.878]
  MoveL 514 to (189.58, -223.38, -18) mm, rotated rx 180 ry 0 rz 179.9 deg; joints [31.307, -31.334, 86.097, -142.959, 59.59, 159.872]
  MoveL 515 to (190.02, -223.28, -18) mm, rotated rx 180 ry 0 rz 179.9 deg; joints [31.297, -31.318, 86.061, -142.964, 59.571, 159.865]
  MoveL 516 to (190.33, -223.19, -18) mm, rotated rx -180 ry 0 rz 179.9 deg; joints [31.289, -31.307, 86.038, -142.969, 59.558, 159.86]
  MoveL 517 to (190.64, -223.07, -18) mm, rotated rx -180 ry 0 rz 179.9 deg; joints [31.28, -31.297, 86.016, -142.974, 59.545, 159.856]
  MoveL 518 to (190.94, -222.93, -18) mm, rotated rx 180 ry 0 rz 179.9 deg; joints [31.27, -31.287, 85.995, -142.98, 59.533, 159.854]
  MoveL 519 to (191.25, -222.77, -18) mm, rotated rx 180 ry 0 rz 179.9 deg; joints [31.26, -31.278, 85.975, -142.988, 59.521, 159.852]
  MoveL 520 to (191.56, -222.57, -18) mm, rotated rx -180 ry 0 rz 179.9 deg; joints [31.249, -31.27, 85.958, -142.997, 59.51, 159.851]
  MoveL 521 to (191.86, -222.34, -18) mm, rotated rx 180 ry 0 rz 179.9 deg; joints [31.236, -31.262, 85.942, -143.007, 59.499, 159.852]
  MoveL 522 to (192.17, -222.08, -18) mm, rotated rx -180 ry 0 rz 179.9 deg; joints [31.223, -31.256, 85.928, -143.019, 59.488, 159.854]
  MoveL 523 to (192.33, -221.92, -18) mm, rotated rx 180 ry 0 rz 179.9 deg; joints [31.216, -31.253, 85.923, -143.026, 59.483, 159.856]
  MoveL 524 to (192.48, -221.76, -18) mm, rotated rx 180 ry 0 rz 179.9 deg; joints [31.208, -31.251, 85.918, -143.033, 59.479, 159.858]
  MoveL 525 to (192.65, -221.55, -18) mm, rotated rx 180 ry 0 rz 179.9 deg; joints [31.199, -31.249, 85.913, -143.042, 59.474, 159.861]
  MoveL 526 to (192.8, -221.34, -18) mm, rotated rx 180 ry 0 rz 179.9 deg; joints [31.19, -31.248, 85.911, -143.052, 59.47, 159.865]
  MoveL 527 to (192.94, -221.13, -18) mm, rotated rx 180 ry 0 rz 179.9 deg; joints [31.182, -31.247, 85.909, -143.061, 59.466, 159.869]
  MoveL 528 to (193.07, -220.92, -18) mm, rotated rx -180 ry 0 rz 179.9 deg; joints [31.173, -31.247, 85.909, -143.07, 59.463, 159.874]
  MoveL 529 to (193.23, -220.62, -18) mm, rotated rx 180 ry 0 rz 179.9 deg; joints [31.161, -31.248, 85.912, -143.083, 59.46, 159.881]
  MoveL 530 to (193.36, -220.31, -18) mm, rotated rx 180 ry 0 rz 179.9 deg; joints [31.15, -31.25, 85.917, -143.097, 59.459, 159.89]
  MoveL 531 to (193.47, -220, -18) mm, rotated rx 180 ry 0 rz 179.9 deg; joints [31.139, -31.253, 85.924, -143.11, 59.458, 159.898]
  MoveL 532 to (193.56, -219.7, -18) mm, rotated rx 180 ry 0 rz 179.9 deg; joints [31.128, -31.257, 85.933, -143.123, 59.458, 159.907]
  MoveL 533 to (193.63, -219.39, -18) mm, rotated rx 180 ry 0 rz 179.9 deg; joints [31.118, -31.262, 85.944, -143.137, 59.46, 159.917]
  MoveL 534 to (193.68, -219.08, -18) mm, rotated rx 180 ry 0 rz 179.9 deg; joints [31.108, -31.267, 85.957, -143.15, 59.462, 159.928]
  MoveL 535 to (193.71, -218.78, -18) mm, rotated rx 180 ry 0 rz 179.9 deg; joints [31.099, -31.274, 85.971, -143.163, 59.465, 159.938]
  MoveL 536 to (193.72, -218.47, -18) mm, rotated rx 180 ry 0 rz 179.9 deg; joints [31.09, -31.281, 85.988, -143.176, 59.47, 159.95]
  MoveL 537 to (193.72, 219.7, -18) mm, rotated rx 180 ry 0 rz 179.9 deg; joints [16.515, -39.025, 103.916, -161.738, 65.07, 172.57]
  MoveL 538 to (193.71, 220, -18) mm, rotated rx 180 ry 0 rz 179.9 deg; joints [16.504, -39.029, 103.925, -161.751, 65.074, 172.577]
  MoveL 539 to (193.68, 220.31, -18) mm, rotated rx 180 ry 0 rz 179.9 deg; joints [16.493, -39.033, 103.936, -161.764, 65.078, 172.584]
  MoveL 540 to (193.62, 220.62, -18) mm, rotated rx 180 ry 0 rz 179.9 deg; joints [16.482, -39.039, 103.949, -161.777, 65.084, 172.591]
  MoveL 541 to (193.55, 220.92, -18) mm, rotated rx 180 ry 0 rz 179.9 deg; joints [16.471, -39.045, 103.963, -161.789, 65.09, 172.599]
  MoveL 542 to (193.48, 221.18, -18) mm, rotated rx -180 ry 0 rz 179.9 deg; joints [16.463, -39.05, 103.976, -161.8, 65.096, 172.605]
  MoveL 543 to (193.39, 221.43, -18) mm, rotated rx 180 ry 0 rz 179.9 deg; joints [16.455, -39.056, 103.991, -161.81, 65.103, 172.612]
  MoveL 544 to (193.29, 221.68, -18) mm, rotated rx -180 ry 0 rz 179.9 deg; joints [16.446, -39.063, 104.007, -161.82, 65.111, 172.619]
  MoveL 545 to (193.16, 221.93, -18) mm, rotated rx 180 ry 0 rz 179.9 deg; joints [16.438, -39.07, 104.024, -161.83, 65.119, 172.626]
  MoveL 546 to (193.02, 222.19, -18) mm, rotated rx 180 ry 0 rz 179.9 deg; joints [16.431, -39.078, 104.043, -161.841, 65.129, 172.633]
  MoveL 547 to (192.86, 222.44, -18) mm, rotated rx -180 ry 0 rz 179.9 deg; joints [16.423, -39.087, 104.064, -161.851, 65.139, 172.64]
  MoveL 548 to (192.68, 222.69, -18) mm, rotated rx -180 ry 0 rz 179.9 deg; joints [16.416, -39.097, 104.087, -161.86, 65.151, 172.648]
  MoveL 549 to (192.48, 222.94, -18) mm, rotated rx 180 ry 0 rz 179.9 deg; joints [16.409, -39.108, 104.112, -161.87, 65.163, 172.656]
  MoveL 550 to (192.27, 223.16, -18) mm, rotated rx 180 ry 0 rz 179.9 deg; joints [16.403, -39.118, 104.136, -161.878, 65.176, 172.663]
  MoveL 551 to (192.04, 223.38, -18) mm, rotated rx -180 ry 0 rz 179.9 deg; joints [16.397, -39.129, 104.162, -161.887, 65.189, 172.671]
  MoveL 552 to (191.79, 223.59, -18) mm, rotated rx -180 ry 0 rz 179.9 deg; joints [16.392, -39.141, 104.19, -161.894, 65.204, 172.679]
  MoveL 553 to (191.54, 223.77, -18) mm, rotated rx -180 ry 0 rz 179.9 deg; joints [16.388, -39.152, 104.217, -161.901, 65.218, 172.686]
  MoveL 554 to (191.28, 223.93, -18) mm, rotated rx 180 ry 0 rz 179.9 deg; joints [16.385, -39.164, 104.243, -161.907, 65.232, 172.692]
  MoveL 555 to (191.03, 224.08, -18) mm, rotated rx -180 ry 0 rz 179.9 deg; joints [16.383, -39.175, 104.269, -161.912, 65.246, 172.699]
  MoveL 556 to (190.78, 224.2, -18) mm, rotated rx -180 ry 0 rz 179.9 deg; joints [16.381, -39.186, 104.295, -161.916, 65.26, 172.704]
  MoveL 557 to (190.53, 224.3, -18) mm, rotated rx 180 ry 0 rz 179.9 deg; joints [16.38, -39.196, 104.32, -161.919, 65.273, 172.71]
  MoveL 558 to (190.28, 224.39, -18) mm, rotated rx 180 ry 0 rz 179.9 deg; joints [16.379, -39.207, 104.345, -161.922, 65.286, 172.715]
  MoveL 559 to (190.02, 224.47, -18) mm, rotated rx -180 ry 0 rz 179.9 deg; joints [16.379, -39.217, 104.369, -161.924, 65.3, 172.72]
  MoveL 560 to (189.72, 224.54, -18) mm, rotated rx 180 ry 0 rz 179.9 deg; joints [16.38, -39.23, 104.398, -161.925, 65.316, 172.725]
  MoveL 561 to (189.41, 224.59, -18) mm, rotated rx -180 ry 0 rz 179.9 deg; joints [16.381, -39.242, 104.426, -161.926, 65.331, 172.73]
  MoveL 562 to (189.1, 224.63, -18) mm, rotated rx 180 ry 0 rz 179.9 deg; joints [16.383, -39.254, 104.454, -161.926, 65.347, 172.734]
  MoveL 563 to (188.8, 224.64, -18) mm, rotated rx 180 ry 0 rz 179.9 deg; joints [16.386, -39.266, 104.482, -161.925, 65.362, 172.739]
  MoveL 564 to (187.57, 224.64, -18) mm, rotated rx -180 ry 0 rz 179.9 deg; joints [16.4, -39.312, 104.59, -161.919, 65.423, 172.754]
  MoveL 565 to (-182.67, 224.64, -18) mm, rotated rx 180 ry 0 rz 179.9 deg; joints [21.725, -50.606, 133.684, -158.091, 82.641, 177.635]
  MoveL 566 to (-188.8, 224.64, -18) mm, rotated rx 180 ry 0 rz 179.9 deg; joints [21.841, -50.747, 134.117, -157.989, 82.917, 177.732]
  MoveL 567 to (-189.1, 224.63, -18) mm, rotated rx -180 ry 0 rz 179.9 deg; joints [21.848, -50.754, 134.138, -157.983, 82.931, 177.737]
  MoveL 568 to (-189.41, 224.59, -18) mm, rotated rx 180 ry 0 rz 179.9 deg; joints [21.855, -50.761, 134.159, -157.976, 82.944, 177.741]
  MoveL 569 to (-189.72, 224.54, -18) mm, rotated rx -180 ry 0 rz 179.9 deg; joints [21.863, -50.767, 134.179, -157.968, 82.957, 177.746]
  MoveL 570 to (-190.02, 224.47, -18) mm, rotated rx 180 ry 0 rz 179.9 deg; joints [21.873, -50.774, 134.199, -157.96, 82.97, 177.75]
  MoveL 571 to (-190.28, 224.39, -18) mm, rotated rx 180 ry 0 rz 179.9 deg; joints [21.881, -50.779, 134.215, -157.952, 82.98, 177.753]
  MoveL 572 to (-190.53, 224.3, -18) mm, rotated rx 180 ry 0 rz 179.9 deg; joints [21.89, -50.784, 134.23, -157.943, 82.99, 177.756]
  MoveL 573 to (-190.78, 224.2, -18) mm, rotated rx -180 ry 0 rz 179.9 deg; joints [21.9, -50.789, 134.245, -157.934, 82.999, 177.758]
  MoveL 574 to (-191.03, 224.08, -18) mm, rotated rx 180 ry 0 rz 179.9 deg; joints [21.91, -50.793, 134.259, -157.923, 83.009, 177.761]
  MoveL 575 to (-191.28, 223.93, -18) mm, rotated rx -180 ry 0 rz 179.9 deg; joints [21.922, -50.798, 134.273, -157.912, 83.018, 177.763]
  MoveL 576 to (-191.54, 223.77, -18) mm, rotated rx 180 ry 0 rz 179.9 deg; joints [21.934, -50.802, 134.286, -157.9, 83.026, 177.765]
  MoveL 577 to (-191.79, 223.59, -18) mm, rotated rx 180 ry 0 rz 179.9 deg; joints [21.948, -50.806, 134.299, -157.887, 83.035, 177.767]
  MoveL 578 to (-192.04, 223.38, -18) mm, rotated rx 180 ry 0 rz 179.9 deg; joints [21.963, -50.81, 134.31, -157.872, 83.043, 177.768]
  MoveL 579 to (-192.27, 223.16, -18) mm, rotated rx -180 ry 0 rz 179.9 deg; joints [21.977, -50.814, 134.32, -157.858, 83.049, 177.769]
  MoveL 580 to (-192.48, 222.94, -18) mm, rotated rx 180 ry 0 rz 179.9 deg; joints [21.991, -50.817, 134.328, -157.844, 83.055, 177.77]
  MoveL 581 to (-192.68, 222.69, -18) mm, rotated rx -180 ry 0 rz 179.9 deg; joints [22.007, -50.819, 134.336, -157.828, 83.06, 177.77]
  MoveL 582 to (-192.86, 222.44, -18) mm, rotated rx 180 ry 0 rz 179.9 deg; joints [22.023, -50.821, 134.342, -157.813, 83.064, 177.77]
  MoveL 583 to (-193.02, 222.19, -18) mm, rotated rx -180 ry 0 rz 179.9 deg; joints [22.038, -50.823, 134.346, -157.798, 83.067, 177.769]
  MoveL 584 to (-193.16, 221.93, -18) mm, rotated rx 180 ry 0 rz 179.9 deg; joints [22.052, -50.824, 134.348, -157.783, 83.069, 177.768]
  MoveL 585 to (-193.29, 221.68, -18) mm, rotated rx 180 ry 0 rz 179.9 deg; joints [22.067, -50.824, 134.35, -157.769, 83.07, 177.767]
  MoveL 586 to (-193.39, 221.43, -18) mm, rotated rx 180 ry 0 rz 179.9 deg; joints [22.081, -50.825, 134.35, -157.755, 83.071, 177.766]
  MoveL 587 to (-193.48, 221.18, -18) mm, rotated rx -180 ry 0 rz 179.9 deg; joints [22.094, -50.825, 134.349, -157.741, 83.071, 177.764]
  MoveL 588 to (-193.55, 220.92, -18) mm, rotated rx 180 ry 0 rz 179.9 deg; joints [22.108, -50.824, 134.347, -157.728, 83.07, 177.762]
  MoveL 589 to (-193.62, 220.62, -18) mm, rotated rx 180 ry 0 rz 179.9 deg; joints [22.123, -50.823, 134.343, -157.712, 83.068, 177.759]
  MoveL 590 to (-193.68, 220.31, -18) mm, rotated rx -180 ry 0 rz 179.9 deg; joints [22.139, -50.822, 134.338, -157.696, 83.065, 177.756]
  MoveL 591 to (-193.71, 220, -18) mm, rotated rx -180 ry 0 rz 179.9 deg; joints [22.154, -50.82, 134.331, -157.68, 83.061, 177.753]
  MoveL 592 to (-193.72, 219.7, -18) mm, rotated rx 180 ry 0 rz 179.9 deg; joints [22.169, -50.817, 134.323, -157.665, 83.057, 177.749]
  MoveL 593 to (-193.72, 216.63, -18) mm, rotated rx -180 ry 0 rz 179.9 deg; joints [22.313, -50.791, 134.235, -157.517, 83.006, 177.71]
  MoveL 594 to (-193.71, 216.32, -18) mm, rotated rx 180 ry 0 rz 179.9 deg; joints [22.328, -50.788, 134.225, -157.502, 83, 177.706]
  MoveL 595 to (-193.67, 216.02, -18) mm, rotated rx 180 ry 0 rz 179.9 deg; joints [22.341, -50.785, 134.214, -157.488, 82.994, 177.701]
  MoveL 596 to (-193.29, 213.56, -18) mm, rotated rx -180 ry 0 rz 179.9 deg; joints [22.449, -50.755, 134.116, -157.376, 82.935, 177.663]
  MoveL 597 to (-192.47, 208.44, -18) mm, rotated rx 180 ry 0 rz 179.9 deg; joints [22.673, -50.692, 133.909, -157.144, 82.813, 177.583]
  MoveL 598 to (-126.66, -206.94, -18) mm, rotated rx -180 ry 0 rz 179.9 deg; joints [37.5, -42.825, 112.257, -140.45, 72.907, 167.284]
  MoveL 599 to (-126.58, -207.4, -18) mm, rotated rx 180 ry 0 rz 179.9 deg; joints [37.513, -42.813, 112.227, -140.433, 72.897, 167.269]
  MoveC 600 to (-127.33, -208.53, -18) mm, rotated rx 180 ry 0 rz 179.9 deg; joints [37.568, -42.811, 112.219, -140.376, 72.905, 167.249] to (-128.52, -207.88, -18) mm, rotated rx 180 ry 0 rz 179.9 deg; joints [37.577, -42.858, 112.335, -140.38, 72.959, 167.292]
  MoveL 601 to (-128.9, -206.76, -18) mm, rotated rx -180 ry 0 rz 179.9 deg; joints [37.55, -42.893, 112.421, -140.417, 72.992, 167.334]
  Set speed (5.6 mm/s)
  MoveL 602 to (-128.9, -206.76, -19.05) mm, rotated rx -180 ry 0 rz 179.9 deg; joints [37.55, -42.831, 112.41, -140.427, 73.032, 167.368]
  MoveC 603 to (-128.61, -206.71, -19.76) mm, rotated rx 180 ry 0 rz 179.9 deg; joints [37.542, -42.782, 112.385, -140.44, 73.048, 167.386] to (-127.91, -206.6, -20.05) mm, rotated rx -180 ry 0 rz 179.9 deg; joints [37.521, -42.747, 112.339, -140.459, 73.036, 167.385]
  Set speed (16.7 mm/s)
  MoveL 604 to (-126.77, -207.43, -20.05) mm, rotated rx 180 ry 0 rz 179.9 deg; joints [37.519, -42.697, 112.217, -140.447, 72.979, 167.337]
  MoveL 605 to (-124.73, -220.31, -20.05) mm, rotated rx 180 ry 0 rz 179.9 deg; joints [37.884, -42.363, 111.39, -139.978, 72.683, 166.903]
  MoveL 606 to (-124.67, -220.62, -20.05) mm, rotated rx 180 ry 0 rz 179.9 deg; joints [37.893, -42.355, 111.369, -139.967, 72.676, 166.893]
  MoveL 607 to (-124.6, -220.92, -20.05) mm, rotated rx 180 ry 0 rz 179.9 deg; joints [37.901, -42.346, 111.348, -139.956, 72.668, 166.882]
  MoveL 608 to (-124.54, -221.13, -20.05) mm, rotated rx 180 ry 0 rz 179.9 deg; joints [37.906, -42.34, 111.333, -139.949, 72.662, 166.874]
  MoveL 609 to (-124.47, -221.34, -20.05) mm, rotated rx 180 ry 0 rz 179.9 deg; joints [37.911, -42.333, 111.317, -139.942, 72.656, 166.866]
  MoveL 610 to (-124.39, -221.54, -20.05) mm, rotated rx 180 ry 0 rz 179.9 deg; joints [37.915, -42.327, 111.301, -139.935, 72.65, 166.859]
  MoveL 611 to (-124.3, -221.75, -20.05) mm, rotated rx -180 ry 0 rz 179.9 deg; joints [37.92, -42.32, 111.283, -139.929, 72.643, 166.85]
  MoveL 612 to (-124.2, -221.95, -20.05) mm, rotated rx 180 ry 0 rz 179.9 deg; joints [37.924, -42.312, 111.265, -139.923, 72.636, 166.842]
  MoveL 613 to (-124.09, -222.16, -20.05) mm, rotated rx -180 ry 0 rz 179.9 deg; joints [37.927, -42.304, 111.246, -139.917, 72.628, 166.834]
  MoveL 614 to (-123.96, -222.36, -20.05) mm, rotated rx -180 ry 0 rz 179.9 deg; joints [37.931, -42.296, 111.227, -139.911, 72.62, 166.825]
  MoveL 615 to (-123.82, -222.57, -20.05) mm, rotated rx -180 ry 0 rz 179.9 deg; joints [37.934, -42.288, 111.206, -139.905, 72.611, 166.816]
  MoveL 616 to (-123.67, -222.77, -20.05) mm, rotated rx 180 ry 0 rz 179.9 deg; joints [37.936, -42.279, 111.184, -139.9, 72.602, 166.806]
  MoveL 617 to (-123.49, -222.97, -20.05) mm, rotated rx -180 ry 0 rz 179.9 deg; joints [37.939, -42.27, 111.161, -139.895, 72.592, 166.796]
  MoveL 618 to (-123.29, -223.19, -20.05) mm, rotated rx 180 ry 0 rz 179.9 deg; joints [37.94, -42.259, 111.136, -139.89, 72.581, 166.786]
  MoveL 619 to (-123.09, -223.38, -20.05) mm, rotated rx -180 ry 0 rz 179.9 deg; joints [37.941, -42.249, 111.111, -139.886, 72.571, 166.776]
  MoveL 620 to (-122.87, -223.56, -20.05) mm, rotated rx -180 ry 0 rz 179.9 deg; joints [37.942, -42.239, 111.087, -139.883, 72.56, 166.766]
  MoveL 621 to (-122.66, -223.72, -20.05) mm, rotated rx -180 ry 0 rz 179.9 deg; joints [37.942, -42.229, 111.063, -139.88, 72.549, 166.757]
  MoveL 622 to (-122.44, -223.86, -20.05) mm, rotated rx 180 ry 0 rz 179.9 deg; joints [37.941, -42.22, 111.041, -139.878, 72.539, 166.748]
  MoveL 623 to (-122.23, -223.99, -20.05) mm, rotated rx 180 ry 0 rz 179.9 deg; joints [37.939, -42.211, 111.019, -139.877, 72.529, 166.74]
  MoveL 624 to (-122.01, -224.11, -20.05) mm, rotated rx 180 ry 0 rz 179.9 deg; joints [37.938, -42.202, 110.998, -139.876, 72.519, 166.732]
  MoveL 625 to (-121.8, -224.21, -20.05) mm, rotated rx -180 ry 0 rz 179.9 deg; joints [37.936, -42.194, 110.978, -139.876, 72.509, 166.725]
  MoveL 626 to (-121.37, -224.37, -20.05) mm, rotated rx -180 ry 0 rz 179.9 deg; joints [37.93, -42.178, 110.939, -139.877, 72.491, 166.711]
  MoveL 627 to (-121.06, -224.47, -20.05) mm, rotated rx 180 ry 0 rz 179.9 deg; joints [37.926, -42.167, 110.913, -139.879, 72.478, 166.702]
  MoveL 628 to (-120.76, -224.54, -20.05) mm, rotated rx 180 ry 0 rz 179.9 deg; joints [37.92, -42.156, 110.888, -139.881, 72.466, 166.694]
  MoveL 629 to (-120.45, -224.59, -20.05) mm, rotated rx -180 ry 0 rz 179.9 deg; joints [37.914, -42.146, 110.864, -139.885, 72.454, 166.686]
  MoveL 630 to (-120.14, -224.62, -20.05) mm, rotated rx -180 ry 0 rz 179.9 deg; joints [37.908, -42.137, 110.841, -139.889, 72.442, 166.679]
  MoveL 631 to (-118.92, -224.64, -20.05) mm, rotated rx 180 ry 0 rz 179.9 deg; joints [37.877, -42.101, 110.755, -139.909, 72.397, 166.654]
  MoveL 632 to (182.67, -224.64, -20.05) mm, rotated rx 180 ry 0 rz 179.9 deg; joints [31.469, -31.498, 86.651, -142.92, 59.957, 160.058]
  MoveL 633 to (188.8, -224.64, -20.05) mm, rotated rx 180 ry 0 rz 179.9 deg; joints [31.359, -31.236, 86.077, -142.93, 59.67, 159.899]
  MoveL 634 to (189.1, -224.62, -20.05) mm, rotated rx -180 ry 0 rz 179.9 deg; joints [31.353, -31.224, 86.049, -142.932, 59.656, 159.891]
  MoveL 635 to (189.41, -224.59, -20.05) mm, rotated rx 180 ry 0 rz 179.9 deg; joints [31.347, -31.211, 86.022, -142.933, 59.642, 159.885]
  MoveL 636 to (189.72, -224.54, -20.05) mm, rotated rx 180 ry 0 rz 179.9 deg; joints [31.34, -31.2, 85.996, -142.936, 59.628, 159.879]
  MoveL 637 to (190.02, -224.46, -20.05) mm, rotated rx -180 ry 0 rz 179.9 deg; joints [31.332, -31.188, 85.972, -142.94, 59.615, 159.873]
  MoveL 638 to (190.27, -224.39, -20.05) mm, rotated rx 180 ry 0 rz 179.9 deg; joints [31.326, -31.179, 85.952, -142.943, 59.604, 159.869]
  MoveL 639 to (190.53, -224.3, -20.05) mm, rotated rx 180 ry 0 rz 179.9 deg; joints [31.318, -31.171, 85.934, -142.947, 59.594, 159.866]
  MoveL 640 to (190.78, -224.19, -20.05) mm, rotated rx 180 ry 0 rz 179.9 deg; joints [31.311, -31.163, 85.916, -142.952, 59.583, 159.864]
  MoveL 641 to (191.03, -224.07, -20.05) mm, rotated rx 180 ry 0 rz 179.9 deg; joints [31.303, -31.155, 85.899, -142.958, 59.573, 159.862]
  MoveL 642 to (191.28, -223.93, -20.05) mm, rotated rx 180 ry 0 rz 179.9 deg; joints [31.294, -31.148, 85.884, -142.964, 59.564, 159.86]
  MoveL 643 to (191.53, -223.77, -20.05) mm, rotated rx 180 ry 0 rz 179.9 deg; joints [31.285, -31.141, 85.869, -142.971, 59.554, 159.86]
  MoveL 644 to (191.78, -223.59, -20.05) mm, rotated rx 180 ry 0 rz 179.9 deg; joints [31.275, -31.135, 85.856, -142.98, 59.545, 159.86]
  MoveL 645 to (192.04, -223.38, -20.05) mm, rotated rx -180 ry 0 rz 179.9 deg; joints [31.264, -31.13, 85.844, -142.989, 59.537, 159.861]
  MoveL 646 to (192.27, -223.16, -20.05) mm, rotated rx -180 ry 0 rz 179.9 deg; joints [31.254, -31.125, 85.835, -142.999, 59.529, 159.864]
  MoveL 647 to (192.48, -222.94, -20.05) mm, rotated rx 180 ry 0 rz 179.9 deg; joints [31.244, -31.122, 85.828, -143.009, 59.523, 159.867]
  MoveL 648 to (192.68, -222.69, -20.05) mm, rotated rx -180 ry 0 rz 179.9 deg; joints [31.233, -31.119, 85.823, -143.02, 59.517, 159.871]
  MoveL 649 to (192.86, -222.44, -20.05) mm, rotated rx 180 ry 0 rz 179.9 deg; joints [31.222, -31.118, 85.82, -143.031, 59.512, 159.875]
  MoveL 650 to (193.02, -222.18, -20.05) mm, rotated rx -180 ry 0 rz 179.9 deg; joints [31.212, -31.118, 85.82, -143.042, 59.508, 159.881]
  MoveL 651 to (193.16, -221.93, -20.05) mm, rotated rx 180 ry 0 rz 179.9 deg; joints [31.202, -31.118, 85.821, -143.053, 59.505, 159.887]
  MoveL 652 to (193.28, -221.68, -20.05) mm, rotated rx 180 ry 0 rz 179.9 deg; joints [31.192, -31.119, 85.824, -143.064, 59.503, 159.893]
  MoveL 653 to (193.39, -221.43, -20.05) mm, rotated rx 180 ry 0 rz 179.9 deg; joints [31.183, -31.121, 85.828, -143.075, 59.502, 159.9]
  MoveL 654 to (193.48, -221.18, -20.05) mm, rotated rx 180 ry 0 rz 179.9 deg; joints [31.174, -31.124, 85.834, -143.086, 59.502, 159.907]
  MoveL 655 to (193.55, -220.92, -20.05) mm, rotated rx 180 ry 0 rz 179.9 deg; joints [31.165, -31.127, 85.842, -143.097, 59.502, 159.915]
  MoveL 656 to (193.62, -220.62, -20.05) mm, rotated rx 180 ry 0 rz 179.9 deg; joints [31.155, -31.132, 85.852, -143.11, 59.503, 159.924]
  MoveL 657 to (193.67, -220.31, -20.05) mm, rotated rx 180 ry 0 rz 179.9 deg; joints [31.145, -31.137, 85.865, -143.123, 59.506, 159.934]
  MoveL 658 to (193.71, -220, -20.05) mm, rotated rx 180 ry 0 rz 179.9 deg; joints [31.136, -31.144, 85.88, -143.137, 59.509, 159.945]
  MoveL 659 to (193.72, -219.7, -20.05) mm, rotated rx -180 ry 0 rz 179.9 deg; joints [31.126, -31.151, 85.896, -143.15, 59.513, 159.956]
  MoveL 660 to (193.72, 219.7, -20.05) mm, rotated rx 180 ry 0 rz 179.9 deg; joints [16.515, -38.913, 103.894, -161.75, 65.156, 172.601]
  MoveL 661 to (193.71, 220, -20.05) mm, rotated rx 180 ry 0 rz 179.9 deg; joints [16.504, -38.916, 103.904, -161.763, 65.16, 172.608]
  MoveL 662 to (193.68, 220.31, -20.05) mm, rotated rx 180 ry 0 rz 179.9 deg; joints [16.493, -38.921, 103.915, -161.776, 65.164, 172.615]
  MoveL 663 to (193.62, 220.62, -20.05) mm, rotated rx -180 ry 0 rz 179.9 deg; joints [16.483, -38.926, 103.927, -161.789, 65.17, 172.622]
  MoveL 664 to (193.55, 220.92, -20.05) mm, rotated rx 180 ry 0 rz 179.9 deg; joints [16.472, -38.932, 103.942, -161.802, 65.176, 172.63]
  MoveL 665 to (193.48, 221.18, -20.05) mm, rotated rx -180 ry 0 rz 179.9 deg; joints [16.464, -38.938, 103.955, -161.812, 65.183, 172.636]
  MoveL 666 to (193.39, 221.43, -20.05) mm, rotated rx 180 ry 0 rz 179.9 deg; joints [16.455, -38.944, 103.969, -161.822, 65.19, 172.643]
  MoveL 667 to (193.29, 221.68, -20.05) mm, rotated rx 180 ry 0 rz 179.9 deg; joints [16.447, -38.951, 103.985, -161.833, 65.197, 172.65]
  MoveL 668 to (193.16, 221.93, -20.05) mm, rotated rx 180 ry 0 rz 179.9 deg; joints [16.439, -38.958, 104.003, -161.843, 65.206, 172.657]
  MoveL 669 to (193.02, 222.19, -20.05) mm, rotated rx -180 ry 0 rz 179.9 deg; joints [16.431, -38.966, 104.022, -161.853, 65.215, 172.664]
  MoveL 670 to (192.86, 222.44, -20.05) mm, rotated rx 180 ry 0 rz 179.9 deg; joints [16.424, -38.975, 104.042, -161.863, 65.225, 172.671]
  MoveL 671 to (192.68, 222.69, -20.05) mm, rotated rx -180 ry 0 rz 179.9 deg; joints [16.416, -38.985, 104.065, -161.873, 65.237, 172.679]
  MoveL 672 to (192.48, 222.94, -20.05) mm, rotated rx -180 ry 0 rz 179.9 deg; joints [16.409, -38.995, 104.09, -161.883, 65.25, 172.687]
  MoveL 673 to (192.27, 223.16, -20.05) mm, rotated rx 180 ry 0 rz 179.9 deg; joints [16.403, -39.005, 104.114, -161.891, 65.262, 172.694]
  MoveL 674 to (192.04, 223.38, -20.05) mm, rotated rx 180 ry 0 rz 179.9 deg; joints [16.398, -39.016, 104.14, -161.899, 65.276, 172.702]
  MoveL 675 to (191.79, 223.59, -20.05) mm, rotated rx 180 ry 0 rz 179.9 deg; joints [16.393, -39.028, 104.168, -161.907, 65.29, 172.709]
  MoveL 676 to (191.54, 223.77, -20.05) mm, rotated rx 180 ry 0 rz 179.9 deg; joints [16.389, -39.04, 104.195, -161.913, 65.304, 172.717]
  MoveL 677 to (191.28, 223.93, -20.05) mm, rotated rx 180 ry 0 rz 179.9 deg; joints [16.386, -39.051, 104.222, -161.919, 65.318, 172.723]
  MoveL 678 to (191.03, 224.08, -20.05) mm, rotated rx -180 ry 0 rz 179.9 deg; joints [16.383, -39.062, 104.248, -161.924, 65.332, 172.729]
  MoveL 679 to (190.78, 224.2, -20.05) mm, rotated rx 180 ry 0 rz 179.9 deg; joints [16.381, -39.073, 104.273, -161.928, 65.346, 172.735]
  MoveL 680 to (190.53, 224.3, -20.05) mm, rotated rx 180 ry 0 rz 179.9 deg; joints [16.38, -39.084, 104.298, -161.931, 65.36, 172.741]
  MoveL 681 to (190.28, 224.39, -20.05) mm, rotated rx 180 ry 0 rz 179.9 deg; joints [16.38, -39.094, 104.323, -161.934, 65.373, 172.746]
  MoveL 682 to (190.02, 224.47, -20.05) mm, rotated rx -180 ry 0 rz 179.9 deg; joints [16.38, -39.105, 104.347, -161.936, 65.386, 172.75]
  MoveL 683 to (189.72, 224.54, -20.05) mm, rotated rx 180 ry 0 rz 179.9 deg; joints [16.38, -39.117, 104.376, -161.937, 65.402, 172.756]
  MoveL 684 to (189.41, 224.59, -20.05) mm, rotated rx -180 ry 0 rz 179.9 deg; joints [16.382, -39.129, 104.405, -161.938, 65.418, 172.761]
  MoveL 685 to (189.1, 224.63, -20.05) mm, rotated rx 180 ry 0 rz 179.9 deg; joints [16.384, -39.141, 104.433, -161.938, 65.433, 172.765]
